LIN {X 0,Y 244.857,Z 831.109,A -85,B 0,C 180,E1 -23796.515,E2 -23796.515} C_VEL
LIN {X 0,Y 244.791,Z 831.344,A -85,B 0,C 180,E1 -23797.056,E2 -23797.056} C_VEL
LIN {X 0,Y 241.341,Z 845.058,A -85,B 0,C 180,E1 -23798.305,E2 -23798.305} C_VEL
LIN {X 0,Y 237.231,Z 858.218,A -85,B 0,C 180,E1 -23799.255,E2 -23799.255} C_VEL
LIN {X 0,Y 231.559,Z 871.694,A -85,B 0,C 180,E1 -23800.015,E2 -23800.015} C_VEL
LIN {X 0,Y 225.914,Z 882.984,A -85,B 0,C 180,E1 -23800.839,E2 -23800.839} C_VEL
LIN {X 0,Y 220.238,Z 892.764,A -85,B 0,C 180,E1 -23801.758,E2 -23801.758} C_VEL
LIN {X 0,Y 213.698,Z 902.652,A -85,B 0,C 180,E1 -23802.963,E2 -23802.963} C_VEL
LIN {X 0,Y 208.1,Z 910.323,A -85,B 0,C 180,E1 -23804.135,E2 -23804.135} C_VEL
LIN {X 0,Y 205.548,Z 913.56,A -85,B 0,C 180,E1 -23804.72,E2 -23804.72} C_VEL
LIN {X 0,Y 202.996,Z 916.447,A -85,B 0,C 180,E1 -23805.095,E2 -23805.095} C_VEL
LIN {X 0,Y 192.619,Z 924.938,A -85,B 0,C 180,E1 -23805.601,E2 -23805.601} C_VEL
LIN {X 0,Y 189.939,Z 927.241,A -85,B 0,C 180,E1 -23806.106,E2 -23806.106} C_VEL
LIN {X 0,Y 181.458,Z 935.069,A -85,B 0,C 180,E1 -23808.816,E2 -23808.816} C_VEL
LIN {X 0,Y 172.726,Z 942.329,A -85,B 0,C 180,E1 -23812.383,E2 -23812.383} C_VEL
LIN {X 0,Y 165.24,Z 947.878,A -85,B 0,C 180,E1 -23816.429,E2 -23816.429} C_VEL
LIN {X 0,Y 159.035,Z 952.034,A -85,B 0,C 180,E1 -23820.911,E2 -23820.911} C_VEL
LIN {X 0,Y 154.257,Z 954.977,A -85,B 0,C 180,E1 -23825.788,E2 -23825.788} C_VEL
LIN {X 0,Y 151.249,Z 956.558,A -85,B 0,C 180,E1 -23831.014,E2 -23831.014} C_VEL
LIN {X 0,Y 149.827,Z 956.906,A -85,B 0,C 180,E1 -23837.294,E2 -23837.294} C_VEL
LIN {X 0,Y 149.411,Z 960.982,A -85,B 0,C 180,E1 -23841.884,E2 -23841.884} C_VEL
LIN {X 0,Y 149.623,Z 962.776,A -85,B 0,C 180,E1 -23844.606,E2 -23844.606} C_VEL
LIN {X 0,Y 149.968,Z 964.104,A -85,B 0,C 180,E1 -23847.31,E2 -23847.31} C_VEL
LIN {X 0,Y 150.384,Z 964.99,A -85,B 0,C 180,E1 -23849.996,E2 -23849.996} C_VEL
LIN {X 0,Y 149.87,Z 965.286,A -85,B 0,C 180,E1 -23852.684,E2 -23852.684} C_VEL
LIN {X 0,Y 149.422,Z 965.12,A -85,B 0,C 180,E1 -23855.394,E2 -23855.394} C_VEL
LIN {X 0,Y 149.11,Z 964.525,A -85,B 0,C 180,E1 -23858.194,E2 -23858.194} C_VEL
LIN {X 0,Y 149.309,Z 962.242,A -85,B 0,C 180,E1 -23863.608,E2 -23863.608} C_VEL
LIN {X 0,Y 150.4,Z 959.454,A -85,B 0,C 180,E1 -23867.678,E2 -23867.678} C_VEL
LIN {X 0,Y 152.856,Z 954.714,A -85,B 0,C 180,E1 -23872.581,E2 -23872.581} C_VEL
LIN {X 0,Y 156.344,Z 949.182,A -85,B 0,C 180,E1 -23876.709,E2 -23876.709} C_VEL
LIN {X 0,Y 160.078,Z 942.88,A -85,B 0,C 180,E1 -23880.32,E2 -23880.32} C_VEL
LIN {X 0,Y 164.723,Z 935.183,A -85,B 0,C 180,E1 -23883.682,E2 -23883.682} C_VEL
LIN {X 0,Y 169.08,Z 927.436,A -85,B 0,C 180,E1 -23886.317,E2 -23886.317} C_VEL
LIN {X 0,Y 173.945,Z 918.156,A -85,B 0,C 180,E1 -23888.769,E2 -23888.769} C_VEL
LIN {X 0,Y 178.68,Z 907.985,A -85,B 0,C 180,E1 -23890.832,E2 -23890.832} C_VEL
LIN {X 0,Y 182.982,Z 896.807,A -85,B 0,C 180,E1 -23892.6,E2 -23892.6} C_VEL
LIN {X 0,Y 186.389,Z 886.413,A -85,B 0,C 180,E1 -23893.851,E2 -23893.851} C_VEL
LIN {X 0,Y 189.626,Z 874.101,A -85,B 0,C 180,E1 -23894.949,E2 -23894.949} C_VEL
LIN {X 0,Y 191.998,Z 861.503,A -85,B 0,C 180,E1 -23895.752,E2 -23895.752} C_VEL
LIN {X 0,Y 193.51,Z 846.926,A -85,B 0,C 180,E1 -23896.366,E2 -23896.366} C_VEL
LIN {X 0,Y 193.334,Z 821.886,A -85,B 0,C 180,E1 -23898.09,E2 -23898.09} C_VEL
LIN {X 0,Y 192.785,Z 805.817,A -85,B 0,C 180,E1 -23899.433,E2 -23899.433} C_VEL
LIN {X 0,Y 190.099,Z 798.147,A -85,B 0,C 180,E1 -23901.251,E2 -23901.251} C_VEL
LIN {X 0,Y 186.949,Z 790.152,A -85,B 0,C 180,E1 -23903.519,E2 -23903.519} C_VEL
LIN {X 0,Y 184.296,Z 784.188,A -85,B 0,C 180,E1 -23905.597,E2 -23905.597} C_VEL
LIN {X 0,Y 181.829,Z 778.84,A -85,B 0,C 180,E1 -23907.744,E2 -23907.744} C_VEL
LIN {X 0,Y 178.972,Z 772.86,A -85,B 0,C 180,E1 -23910.603,E2 -23910.603} C_VEL
LIN {X 0,Y 175.032,Z 765.017,A -85,B 0,C 180,E1 -23915.66,E2 -23915.66} C_VEL
LIN {X 0,Y 172.015,Z 759.221,A -85,B 0,C 180,E1 -23921.926,E2 -23921.926} C_VEL
LIN {X 0,Y 171.237,Z 756.818,A -85,B 0,C 180,E1 -23925.744,E2 -23925.744} C_VEL
LIN {X 0,Y 171.154,Z 756.438,A -85,B 0,C 180,E1 -23930.547,E2 -23930.547} C_VEL
LIN {X 0,Y 173.798,Z 758.074,A -85,B 0,C 180,E1 -23938.487,E2 -23938.487} C_VEL
LIN {X 0,Y 175.332,Z 761.318,A -85,B 0,C 180,E1 -23941.273,E2 -23941.273} C_VEL
LIN {X 0,Y 177.527,Z 763.638,A -85,B 0,C 180,E1 -23944.097,E2 -23944.097} C_VEL
LIN {X 0,Y 179.95,Z 767.21,A -85,B 0,C 180,E1 -23946.729,E2 -23946.729} C_VEL
LIN {X 0,Y 183.962,Z 773.224,A -85,B 0,C 180,E1 -23950.335,E2 -23950.335} C_VEL
LIN {X 0,Y 186.785,Z 777.685,A -85,B 0,C 180,E1 -23952.504,E2 -23952.504} C_VEL
LIN {X 0,Y 190.835,Z 784.368,A -85,B 0,C 180,E1 -23955.234,E2 -23955.234} C_VEL
LIN {X 0,Y 195.08,Z 792.248,A -85,B 0,C 180,E1 -23957.807,E2 -23957.807} C_VEL
LIN {X 0,Y 197.268,Z 796.713,A -85,B 0,C 180,E1 -23959.024,E2 -23959.024} C_VEL
LIN {X 0,Y 195.596,Z 824.391,A -85,B 0,C 180,E1 -23960.277,E2 -23960.277} C_VEL
LIN {X 0,Y 194.043,Z 837.391,A -85,B 0,C 180,E1 -23961.235,E2 -23961.235} C_VEL
LIN {X 0,Y 191.694,Z 849.84,A -85,B 0,C 180,E1 -23962.515,E2 -23962.515} C_VEL
LIN {X 0,Y 188.741,Z 860.968,A -85,B 0,C 180,E1 -23964.019,E2 -23964.019} C_VEL
LIN {X 0,Y 184.831,Z 872.603,A -85,B 0,C 180,E1 -23966.071,E2 -23966.071} C_VEL
LIN {X 0,Y 180.804,Z 882.425,A -85,B 0,C 180,E1 -23968.287,E2 -23968.287} C_VEL
LIN {X 0,Y 176.714,Z 890.906,A -85,B 0,C 180,E1 -23970.72,E2 -23970.72} C_VEL
LIN {X 0,Y 172.62,Z 898.364,A -85,B 0,C 180,E1 -23973.43,E2 -23973.43} C_VEL
LIN {X 0,Y 168.723,Z 904.617,A -85,B 0,C 180,E1 -23976.28,E2 -23976.28} C_VEL
LIN {X 0,Y 164.664,Z 910.533,A -85,B 0,C 180,E1 -23979.809,E2 -23979.809} C_VEL
LIN {X 0,Y 160.835,Z 915.42,A -85,B 0,C 180,E1 -23983.712,E2 -23983.712} C_VEL
LIN {X 0,Y 157.431,Z 919.174,A -85,B 0,C 180,E1 -23987.967,E2 -23987.967} C_VEL
LIN {X 0,Y 155.666,Z 920.852,A -85,B 0,C 180,E1 -23990.802,E2 -23990.802} C_VEL
LIN {X 0,Y 153.445,Z 922.533,A -85,B 0,C 180,E1 -23995.532,E2 -23995.532} C_VEL
LIN {X 0,Y 152.21,Z 922.921,A -85,B 0,C 180,E1 -23999.481,E2 -23999.481} C_VEL
LIN {X 0,Y 151.648,Z 922.674,A -85,B 0,C 180,E1 -24002.395,E2 -24002.395} C_VEL
LIN {X 0,Y 151.373,Z 921.923,A -85,B 0,C 180,E1 -24005.305,E2 -24005.305} C_VEL
LIN {X 0,Y 151.422,Z 920.718,A -85,B 0,C 180,E1 -24008.208,E2 -24008.208} C_VEL
LIN {X 0,Y 152.006,Z 918.04,A -85,B 0,C 180,E1 -24012.515,E2 -24012.515} C_VEL
LIN {X 0,Y 153.266,Z 914.247,A -85,B 0,C 180,E1 -24016.75,E2 -24016.75} C_VEL
LIN {X 0,Y 155.055,Z 909.269,A -85,B 0,C 180,E1 -24020.876,E2 -24020.876} C_VEL
LIN {X 0,Y 157.321,Z 902.95,A -85,B 0,C 180,E1 -24024.878,E2 -24024.878} C_VEL
LIN {X 0,Y 160.173,Z 895.068,A -85,B 0,C 180,E1 -24028.747,E2 -24028.747} C_VEL
LIN {X 0,Y 163.015,Z 886.699,A -85,B 0,C 180,E1 -24031.983,E2 -24031.983} C_VEL
LIN {X 0,Y 166.212,Z 876.183,A -85,B 0,C 180,E1 -24035.159,E2 -24035.159} C_VEL
LIN {X 0,Y 169.239,Z 864.857,A -85,B 0,C 180,E1 -24037.82,E2 -24037.82} C_VEL
LIN {X 0,Y 171.631,Z 854.357,A -85,B 0,C 180,E1 -24039.728,E2 -24039.728} C_VEL
LIN {X 0,Y 173.863,Z 841.585,A -85,B 0,C 180,E1 -24041.516,E2 -24041.516} C_VEL
LIN {X 0,Y 175.492,Z 828.533,A -85,B 0,C 180,E1 -24042.846,E2 -24042.846} C_VEL
LIN {X 0,Y 176.383,Z 815.217,A -85,B 0,C 180,E1 -24043.746,E2 -24043.746} C_VEL
LIN {X 0,Y 177.602,Z 782.378,A -85,B 0,C 180,E1 -24045.194,E2 -24045.194} C_VEL
LIN {X 0,Y 172.041,Z 770.25,A -85,B 0,C 180,E1 -24047.17,E2 -24047.17} C_VEL
LIN {X 0,Y 163.489,Z 754.986,A -85,B 0,C 180,E1 -24050.347,E2 -24050.347} C_VEL
LIN {X 0,Y 157.596,Z 745.662,A -85,B 0,C 180,E1 -24052.739,E2 -24052.739} C_VEL
LIN {X 0,Y 155.084,Z 741.988,A -85,B 0,C 180,E1 -24053.801,E2 -24053.801} C_VEL
LIN {X 0,Y 152.506,Z 738.118,A -85,B 0,C 180,E1 -24054.953,E2 -24054.953} C_VEL
LIN {X 0,Y 150.687,Z 735.478,A -85,B 0,C 180,E1 -24055.813,E2 -24055.813} C_VEL
LIN {X 0,Y 150.305,Z 734.187,A -85,B 0,C 180,E1 -24056.285,E2 -24056.285} C_VEL
LIN {X 0,Y 150.188,Z 733.748,A -85,B 0,C 180,E1 -24057.238,E2 -24057.238} C_VEL
LIN {X 0,Y 150.208,Z 733.739,A -85,B 0,C 180,E1 -24062.627,E2 -24062.627} C_VEL
LIN {X 0,Y 150.176,Z 733.747,A -85,B 0,C 180,E1 -24067.477,E2 -24067.477} C_VEL
LIN {X 0,Y 150.21,Z 733.927,A -85,B 0,C 180,E1 -24072.797,E2 -24072.797} C_VEL
LIN {X 0,Y 150.427,Z 734.862,A -85,B 0,C 180,E1 -24073.238,E2 -24073.238} C_VEL
LIN {X 0,Y 161.112,Z 767.276,A -85,B 0,C 180,E1 -24076.72,E2 -24076.72} C_VEL
LIN {X 0,Y 158.692,Z 816.623,A -85,B 0,C 180,E1 -24080.253,E2 -24080.253} C_VEL
LIN {X 0,Y 157.835,Z 828.145,A -85,B 0,C 180,E1 -24081.435,E2 -24081.435} C_VEL
LIN {X 0,Y 156.889,Z 838.329,A -85,B 0,C 180,E1 -24082.789,E2 -24082.789} C_VEL
LIN {X 0,Y 155.794,Z 848.57,A -85,B 0,C 180,E1 -24084.477,E2 -24084.477} C_VEL
LIN {X 0,Y 154.801,Z 857.302,A -85,B 0,C 180,E1 -24086.209,E2 -24086.209} C_VEL
LIN {X 0,Y 153.773,Z 866.172,A -85,B 0,C 180,E1 -24088.291,E2 -24088.291} C_VEL
LIN {X 0,Y 152.724,Z 874.335,A -85,B 0,C 180,E1 -24090.545,E2 -24090.545} C_VEL
LIN {X 0,Y 151.782,Z 882.385,A -85,B 0,C 180,E1 -24093.162,E2 -24093.162} C_VEL
LIN {X 0,Y 150.909,Z 891.404,A -85,B 0,C 180,E1 -24096.68,E2 -24096.68} C_VEL
LIN {X 0,Y 150.428,Z 898.5,A -85,B 0,C 180,E1 -24099.969,E2 -24099.969} C_VEL
LIN {X 0,Y 150.233,Z 904.129,A -85,B 0,C 180,E1 -24102.999,E2 -24102.999} C_VEL
LIN {X 0,Y 150.402,Z 909.603,A -85,B 0,C 180,E1 -24106.488,E2 -24106.488} C_VEL
LIN {X 0,Y 151.263,Z 914.934,A -85,B 0,C 180,E1 -24110.641,E2 -24110.641} C_VEL
LIN {X 0,Y 152.752,Z 919.142,A -85,B 0,C 180,E1 -24114.72,E2 -24114.72} C_VEL
LIN {X 0,Y 154.695,Z 922.06,A -85,B 0,C 180,E1 -24118.284,E2 -24118.284} C_VEL
LIN {X 0,Y 157.752,Z 924.553,A -85,B 0,C 180,E1 -24122.553,E2 -24122.553} C_VEL
LIN {X 0,Y 162.55,Z 926.08,A -85,B 0,C 180,E1 -24127.452,E2 -24127.452} C_VEL
LIN {X 0,Y 165.353,Z 926.213,A -85,B 0,C 180,E1 -24129.788,E2 -24129.788} C_VEL
LIN {X 0,Y 171.747,Z 925.212,A -85,B 0,C 180,E1 -24134.213,E2 -24134.213} C_VEL
LIN {X 0,Y 176.15,Z 923.903,A -85,B 0,C 180,E1 -24136.745,E2 -24136.745} C_VEL
LIN {X 0,Y 183.164,Z 920.704,A -85,B 0,C 180,E1 -24140.202,E2 -24140.202} C_VEL
LIN {X 0,Y 189.495,Z 916.99,A -85,B 0,C 180,E1 -24142.919,E2 -24142.919} C_VEL
LIN {X 0,Y 196.24,Z 912.131,A -85,B 0,C 180,E1 -24145.452,E2 -24145.452} C_VEL
LIN {X 0,Y 202.2,Z 907.143,A -85,B 0,C 180,E1 -24147.422,E2 -24147.422} C_VEL
LIN {X 0,Y 208.317,Z 901.17,A -85,B 0,C 180,E1 -24149.287,E2 -24149.287} C_VEL
LIN {X 0,Y 214.931,Z 893.757,A -85,B 0,C 180,E1 -24151.12,E2 -24151.12} C_VEL
LIN {X 0,Y 220.31,Z 886.741,A -85,B 0,C 180,E1 -24152.506,E2 -24152.506} C_VEL
LIN {X 0,Y 225.718,Z 878.716,A -85,B 0,C 180,E1 -24153.818,E2 -24153.818} C_VEL
LIN {X 0,Y 231.039,Z 869.384,A -85,B 0,C 180,E1 -24155.041,E2 -24155.041} C_VEL
LIN {X 0,Y 236.282,Z 858.337,A -85,B 0,C 180,E1 -24156.239,E2 -24156.239} C_VEL
LIN {X 0,Y 238.914,Z 851.646,A -85,B 0,C 180,E1 -24156.816,E2 -24156.816} C_VEL
LIN {X 0,Y 238.877,Z 851.821,A -85,B 0,C 180,E1 -24157.057,E2 -24157.057} C_VEL
LIN {X 0,Y 236.308,Z 858.808,A -85,B 0,C 180,E1 -24157.555,E2 -24157.555} C_VEL
LIN {X 0,Y 230.506,Z 871.836,A -85,B 0,C 180,E1 -24158.266,E2 -24158.266} C_VEL
LIN {X 0,Y 224.981,Z 882.268,A -85,B 0,C 180,E1 -24158.984,E2 -24158.984} C_VEL
LIN {X 0,Y 218.731,Z 892.42,A -85,B 0,C 180,E1 -24159.9,E2 -24159.9} C_VEL
LIN {X 0,Y 212.695,Z 901.133,A -85,B 0,C 180,E1 -24160.896,E2 -24160.896} C_VEL
LIN {X 0,Y 206.139,Z 909.58,A -85,B 0,C 180,E1 -24162.134,E2 -24162.134} C_VEL
LIN {X 0,Y 199.226,Z 917.636,A -85,B 0,C 180,E1 -24163.679,E2 -24163.679} C_VEL
LIN {X 0,Y 192.57,Z 924.669,A -85,B 0,C 180,E1 -24165.364,E2 -24165.364} C_VEL
LIN {X 0,Y 189.939,Z 927.241,A -85,B 0,C 180,E1 -24166.106,E2 -24166.106} C_VEL
LIN {X 0,Y 186.072,Z 930.673,A -85,B 0,C 180,E1 -24167.018,E2 -24167.018} C_VEL
LIN {X 0,Y 178.445,Z 935.858,A -85,B 0,C 180,E1 -24168.222,E2 -24168.222} C_VEL
LIN {X 0,Y 170.825,Z 940.29,A -85,B 0,C 180,E1 -24169.663,E2 -24169.663} C_VEL
LIN {X 0,Y 167.047,Z 942.549,A -85,B 0,C 180,E1 -24170.951,E2 -24170.951} C_VEL
LIN {X 0,Y 161.211,Z 946.474,A -85,B 0,C 180,E1 -24173.943,E2 -24173.943} C_VEL
LIN {X 0,Y 155.936,Z 949.734,A -85,B 0,C 180,E1 -24177.255,E2 -24177.255} C_VEL
LIN {X 0,Y 150.174,Z 952.868,A -85,B 0,C 180,E1 -24182.092,E2 -24182.092} C_VEL
LIN {X 0,Y 147.802,Z 953.95,A -85,B 0,C 180,E1 -24184.658,E2 -24184.658} C_VEL
LIN {X 0,Y 144.57,Z 955.216,A -85,B 0,C 180,E1 -24190.101,E2 -24190.101} C_VEL
LIN {X 0,Y 142.969,Z 955.384,A -85,B 0,C 180,E1 -24196.493,E2 -24196.493} C_VEL
LIN {X 0,Y 142.387,Z 959.731,A -85,B 0,C 180,E1 -24201.48,E2 -24201.48} C_VEL
LIN {X 0,Y 142.55,Z 961.596,A -85,B 0,C 180,E1 -24204.337,E2 -24204.337} C_VEL
LIN {X 0,Y 142.893,Z 962.963,A -85,B 0,C 180,E1 -24207.177,E2 -24207.177} C_VEL
LIN {X 0,Y 143.334,Z 963.887,A -85,B 0,C 180,E1 -24209.996,E2 -24209.996} C_VEL
LIN {X 0,Y 142.793,Z 964.216,A -85,B 0,C 180,E1 -24212.817,E2 -24212.817} C_VEL
LIN {X 0,Y 142.343,Z 964.109,A -85,B 0,C 180,E1 -24215.663,E2 -24215.663} C_VEL
LIN {X 0,Y 142.035,Z 963.562,A -85,B 0,C 180,E1 -24218.532,E2 -24218.532} C_VEL
LIN {X 0,Y 142.361,Z 961.325,A -85,B 0,C 180,E1 -24224.286,E2 -24224.286} C_VEL
LIN {X 0,Y 143.585,Z 958.615,A -85,B 0,C 180,E1 -24228.547,E2 -24228.547} C_VEL
LIN {X 0,Y 145.66,Z 954.974,A -85,B 0,C 180,E1 -24232.701,E2 -24232.701} C_VEL
LIN {X 0,Y 148.805,Z 950.346,A -85,B 0,C 180,E1 -24236.654,E2 -24236.654} C_VEL
LIN {X 0,Y 153.212,Z 943.497,A -85,B 0,C 180,E1 -24241.063,E2 -24241.063} C_VEL
LIN {X 0,Y 158.008,Z 936.183,A -85,B 0,C 180,E1 -24244.544,E2 -24244.544} C_VEL
LIN {X 0,Y 163.423,Z 927.179,A -85,B 0,C 180,E1 -24247.789,E2 -24247.789} C_VEL
LIN {X 0,Y 169.016,Z 917.092,A -85,B 0,C 180,E1 -24250.515,E2 -24250.515} C_VEL
LIN {X 0,Y 173.916,Z 906.962,A -85,B 0,C 180,E1 -24252.595,E2 -24252.595} C_VEL
LIN {X 0,Y 178.438,Z 895.826,A -85,B 0,C 180,E1 -24254.35,E2 -24254.35} C_VEL
LIN {X 0,Y 181.987,Z 885.454,A -85,B 0,C 180,E1 -24255.592,E2 -24255.592} C_VEL
LIN {X 0,Y 185.228,Z 873.548,A -85,B 0,C 180,E1 -24256.663,E2 -24256.663} C_VEL
LIN {X 0,Y 187.809,Z 860.468,A -85,B 0,C 180,E1 -24257.497,E2 -24257.497} C_VEL
LIN {X 0,Y 189.23,Z 847.787,A -85,B 0,C 180,E1 -24258.047,E2 -24258.047} C_VEL
LIN {X 0,Y 189.256,Z 823.547,A -85,B 0,C 180,E1 -24259.752,E2 -24259.752} C_VEL
LIN {X 0,Y 188.922,Z 808.906,A -85,B 0,C 180,E1 -24261.006,E2 -24261.006} C_VEL
LIN {X 0,Y 185.667,Z 799.516,A -85,B 0,C 180,E1 -24263.439,E2 -24263.439} C_VEL
LIN {X 0,Y 182.075,Z 790.42,A -85,B 0,C 180,E1 -24266.427,E2 -24266.427} C_VEL
LIN {X 0,Y 179.383,Z 784.402,A -85,B 0,C 180,E1 -24268.929,E2 -24268.929} C_VEL
LIN {X 0,Y 176.895,Z 778.825,A -85,B 0,C 180,E1 -24271.681,E2 -24271.681} C_VEL
LIN {X 0,Y 173.526,Z 771.565,A -85,B 0,C 180,E1 -24276.427,E2 -24276.427} C_VEL
LIN {X 0,Y 170.856,Z 765.951,A -85,B 0,C 180,E1 -24282.572,E2 -24282.572} C_VEL
LIN {X 0,Y 170.254,Z 763.802,A -85,B 0,C 180,E1 -24286.045,E2 -24286.045} C_VEL
LIN {X 0,Y 170.397,Z 763.591,A -85,B 0,C 180,E1 -24291.813,E2 -24291.813} C_VEL
LIN {X 0,Y 172.553,Z 764.994,A -85,B 0,C 180,E1 -24297.97,E2 -24297.97} C_VEL
LIN {X 0,Y 174.128,Z 768.299,A -85,B 0,C 180,E1 -24300.973,E2 -24300.973} C_VEL
LIN {X 0,Y 175.954,Z 770.323,A -85,B 0,C 180,E1 -24303.432,E2 -24303.432} C_VEL
LIN {X 0,Y 178.897,Z 774.892,A -85,B 0,C 180,E1 -24306.769,E2 -24306.769} C_VEL
LIN {X 0,Y 181.863,Z 779.533,A -85,B 0,C 180,E1 -24309.55,E2 -24309.55} C_VEL
LIN {X 0,Y 185.516,Z 785.499,A -85,B 0,C 180,E1 -24312.449,E2 -24312.449} C_VEL
LIN {X 0,Y 190.41,Z 794.409,A -85,B 0,C 180,E1 -24315.798,E2 -24315.798} C_VEL
LIN {X 0,Y 193.002,Z 799.778,A -85,B 0,C 180,E1 -24317.418,E2 -24317.418} C_VEL
LIN {X 0,Y 191.339,Z 825.631,A -85,B 0,C 180,E1 -24318.63,E2 -24318.63} C_VEL
LIN {X 0,Y 189.639,Z 839.007,A -85,B 0,C 180,E1 -24319.64,E2 -24319.64} C_VEL
LIN {X 0,Y 187.173,Z 851.209,A -85,B 0,C 180,E1 -24320.914,E2 -24320.914} C_VEL
LIN {X 0,Y 183.996,Z 862.479,A -85,B 0,C 180,E1 -24322.456,E2 -24322.456} C_VEL
LIN {X 0,Y 180.29,Z 873.055,A -85,B 0,C 180,E1 -24324.338,E2 -24324.338} C_VEL
LIN {X 0,Y 176.046,Z 882.97,A -85,B 0,C 180,E1 -24326.568,E2 -24326.568} C_VEL
LIN {X 0,Y 171.264,Z 892.376,A -85,B 0,C 180,E1 -24329.309,E2 -24329.309} C_VEL
LIN {X 0,Y 166.475,Z 900.52,A -85,B 0,C 180,E1 -24332.407,E2 -24332.407} C_VEL
LIN {X 0,Y 162.055,Z 907.056,A -85,B 0,C 180,E1 -24335.602,E2 -24335.602} C_VEL
LIN {X 0,Y 157.839,Z 912.736,A -85,B 0,C 180,E1 -24339.291,E2 -24339.291} C_VEL
LIN {X 0,Y 153.986,Z 917.204,A -85,B 0,C 180,E1 -24343.206,E2 -24343.206} C_VEL
LIN {X 0,Y 151.683,Z 919.544,A -85,B 0,C 180,E1 -24345.979,E2 -24345.979} C_VEL
LIN {X 0,Y 149.656,Z 921.439,A -85,B 0,C 180,E1 -24348.9,E2 -24348.9} C_VEL
LIN {X 0,Y 147.959,Z 922.759,A -85,B 0,C 180,E1 -24351.872,E2 -24351.872} C_VEL
LIN {X 0,Y 146.615,Z 923.598,A -85,B 0,C 180,E1 -24354.89,E2 -24354.89} C_VEL
LIN {X 0,Y 145.575,Z 923.958,A -85,B 0,C 180,E1 -24357.929,E2 -24357.929} C_VEL
LIN {X 0,Y 144.831,Z 923.822,A -85,B 0,C 180,E1 -24360.976,E2 -24360.976} C_VEL
LIN {X 0,Y 144.416,Z 923.251,A -85,B 0,C 180,E1 -24364.029,E2 -24364.029} C_VEL
LIN {X 0,Y 144.361,Z 921.921,A -85,B 0,C 180,E1 -24367.668,E2 -24367.668} C_VEL
LIN {X 0,Y 145.083,Z 918.687,A -85,B 0,C 180,E1 -24373.108,E2 -24373.108} C_VEL
LIN {X 0,Y 146.441,Z 914.74,A -85,B 0,C 180,E1 -24377.532,E2 -24377.532} C_VEL
LIN {X 0,Y 148.376,Z 909.584,A -85,B 0,C 180,E1 -24381.835,E2 -24381.835} C_VEL
LIN {X 0,Y 150.838,Z 903.098,A -85,B 0,C 180,E1 -24385.996,E2 -24385.996} C_VEL
LIN {X 0,Y 153.888,Z 895.031,A -85,B 0,C 180,E1 -24390.004,E2 -24390.004} C_VEL
LIN {X 0,Y 156.754,Z 886.775,A -85,B 0,C 180,E1 -24393.217,E2 -24393.217} C_VEL
LIN {X 0,Y 159.938,Z 876.714,A -85,B 0,C 180,E1 -24396.311,E2 -24396.311} C_VEL
LIN {X 0,Y 162.815,Z 866.371,A -85,B 0,C 180,E1 -24398.818,E2 -24398.818} C_VEL
LIN {X 0,Y 165.688,Z 854.358,A -85,B 0,C 180,E1 -24401.047,E2 -24401.047} C_VEL
LIN {X 0,Y 167.901,Z 842.082,A -85,B 0,C 180,E1 -24402.79,E2 -24402.79} C_VEL
LIN {X 0,Y 169.575,Z 829.05,A -85,B 0,C 180,E1 -24404.134,E2 -24404.134} C_VEL
LIN {X 0,Y 170.521,Z 815.506,A -85,B 0,C 180,E1 -24405.055,E2 -24405.055} C_VEL
LIN {X 0,Y 171.772,Z 784.662,A -85,B 0,C 180,E1 -24406.448,E2 -24406.448} C_VEL
LIN {X 0,Y 166.895,Z 773.878,A -85,B 0,C 180,E1 -24408.295,E2 -24408.295} C_VEL
LIN {X 0,Y 158.208,Z 758.184,A -85,B 0,C 180,E1 -24411.745,E2 -24411.745} C_VEL
LIN {X 0,Y 151.544,Z 747.775,A -85,B 0,C 180,E1 -24414.639,E2 -24414.639} C_VEL
LIN {X 0,Y 148.161,Z 742.893,A -85,B 0,C 180,E1 -24416.227,E2 -24416.227} C_VEL
LIN {X 0,Y 145.883,Z 739.368,A -85,B 0,C 180,E1 -24417.383,E2 -24417.383} C_VEL
LIN {X 0,Y 143.969,Z 737.259,A -85,B 0,C 180,E1 -24418.336,E2 -24418.336} C_VEL
LIN {X 0,Y 143.173,Z 735.183,A -85,B 0,C 180,E1 -24419.065,E2 -24419.065} C_VEL
LIN {X 0,Y 143.096,Z 734.694,A -85,B 0,C 180,E1 -24419.825,E2 -24419.825} C_VEL
LIN {X 0,Y 143.14,Z 734.61,A -85,B 0,C 180,E1 -24423.416,E2 -24423.416} C_VEL
LIN {X 0,Y 143.065,Z 734.665,A -85,B 0,C 180,E1 -24429.694,E2 -24429.694} C_VEL
LIN {X 0,Y 143.169,Z 734.859,A -85,B 0,C 180,E1 -24432.164,E2 -24432.164} C_VEL
LIN {X 0,Y 143.327,Z 735.632,A -85,B 0,C 180,E1 -24432.545,E2 -24432.545} C_VEL
LIN {X 0,Y 154.136,Z 768.162,A -85,B 0,C 180,E1 -24436.231,E2 -24436.231} C_VEL
LIN {X 0,Y 151.652,Z 816.898,A -85,B 0,C 180,E1 -24439.874,E2 -24439.874} C_VEL
LIN {X 0,Y 150.738,Z 829.345,A -85,B 0,C 180,E1 -24441.206,E2 -24441.206} C_VEL
LIN {X 0,Y 149.781,Z 839.313,A -85,B 0,C 180,E1 -24442.598,E2 -24442.598} C_VEL
LIN {X 0,Y 148.649,Z 849.364,A -85,B 0,C 180,E1 -24444.341,E2 -24444.341} C_VEL
LIN {X 0,Y 147.539,Z 859.005,A -85,B 0,C 180,E1 -24446.374,E2 -24446.374} C_VEL
LIN {X 0,Y 146.39,Z 868.536,A -85,B 0,C 180,E1 -24448.788,E2 -24448.788} C_VEL
LIN {X 0,Y 145.249,Z 877.393,A -85,B 0,C 180,E1 -24451.457,E2 -24451.457} C_VEL
LIN {X 0,Y 144.441,Z 884.715,A -85,B 0,C 180,E1 -24454.029,E2 -24454.029} C_VEL
LIN {X 0,Y 143.651,Z 892.968,A -85,B 0,C 180,E1 -24457.44,E2 -24457.44} C_VEL
LIN {X 0,Y 143.273,Z 899.543,A -85,B 0,C 180,E1 -24460.663,E2 -24460.663} C_VEL
LIN {X 0,Y 143.14,Z 905.903,A -85,B 0,C 180,E1 -24464.333,E2 -24464.333} C_VEL
LIN {X 0,Y 143.575,Z 911.628,A -85,B 0,C 180,E1 -24468.256,E2 -24468.256} C_VEL
LIN {X 0,Y 144.411,Z 915.811,A -85,B 0,C 180,E1 -24471.604,E2 -24471.604} C_VEL
LIN {X 0,Y 146.117,Z 920.106,A -85,B 0,C 180,E1 -24475.862,E2 -24475.862} C_VEL
LIN {X 0,Y 148.485,Z 923.397,A -85,B 0,C 180,E1 -24480,E2 -24480} C_VEL
LIN {X 0,Y 152.814,Z 926.294,A -85,B 0,C 180,E1 -24485.277,E2 -24485.277} C_VEL
LIN {X 0,Y 156.431,Z 927.329,A -85,B 0,C 180,E1 -24488.714,E2 -24488.714} C_VEL
LIN {X 0,Y 161.463,Z 927.53,A -85,B 0,C 180,E1 -24492.57,E2 -24492.57} C_VEL
LIN {X 0,Y 164.908,Z 927.235,A -85,B 0,C 180,E1 -24494.815,E2 -24494.815} C_VEL
LIN {X 0,Y 172.527,Z 925.233,A -85,B 0,C 180,E1 -24499.019,E2 -24499.019} C_VEL
LIN {X 0,Y 178.85,Z 922.67,A -85,B 0,C 180,E1 -24501.919,E2 -24501.919} C_VEL
LIN {X 0,Y 185.553,Z 919.115,A -85,B 0,C 180,E1 -24504.622,E2 -24504.622} C_VEL
LIN {X 0,Y 192.667,Z 914.465,A -85,B 0,C 180,E1 -24507.127,E2 -24507.127} C_VEL
LIN {X 0,Y 200.161,Z 908.58,A -85,B 0,C 180,E1 -24509.443,E2 -24509.443} C_VEL
LIN {X 0,Y 205.326,Z 903.977,A -85,B 0,C 180,E1 -24510.892,E2 -24510.892} C_VEL
LIN {X 0,Y 211.943,Z 897.119,A -85,B 0,C 180,E1 -24512.605,E2 -24512.605} C_VEL
LIN {X 0,Y 218.691,Z 888.993,A -85,B 0,C 180,E1 -24514.221,E2 -24514.221} C_VEL
LIN {X 0,Y 224.581,Z 880.679,A -85,B 0,C 180,E1 -24515.543,E2 -24515.543} C_VEL
LIN {X 0,Y 228.365,Z 874.777,A -85,B 0,C 180,E1 -24516.316,E2 -24516.316} C_VEL
LIN {X 0,Y 227.941,Z 875.72,A -85,B 0,C 180,E1 -24516.709,E2 -24516.709} C_VEL
LIN {X 0,Y 220.701,Z 887.61,A -85,B 0,C 180,E1 -24517.59,E2 -24517.59} C_VEL
LIN {X 0,Y 213.56,Z 897.825,A -85,B 0,C 180,E1 -24518.59,E2 -24518.59} C_VEL
LIN {X 0,Y 205.949,Z 907.304,A -85,B 0,C 180,E1 -24519.838,E2 -24519.838} C_VEL
LIN {X 0,Y 198.644,Z 915.456,A -85,B 0,C 180,E1 -24521.247,E2 -24521.247} C_VEL
LIN {X 0,Y 190.336,Z 923.726,A -85,B 0,C 180,E1 -24523.172,E2 -24523.172} C_VEL
LIN {X 0,Y 182.45,Z 930.784,A -85,B 0,C 180,E1 -24525.328,E2 -24525.328} C_VEL
LIN {X 0,Y 176.206,Z 935.857,A -85,B 0,C 180,E1 -24527.304,E2 -24527.304} C_VEL
LIN {X 0,Y 169.372,Z 941.038,A -85,B 0,C 180,E1 -24529.968,E2 -24529.968} C_VEL
LIN {X 0,Y 167.047,Z 942.549,A -85,B 0,C 180,E1 -24530.951,E2 -24530.951} C_VEL
LIN {X 0,Y 163.342,Z 944.808,A -85,B 0,C 180,E1 -24532.373,E2 -24532.373} C_VEL
LIN {X 0,Y 156.022,Z 947.759,A -85,B 0,C 180,E1 -24534.534,E2 -24534.534} C_VEL
LIN {X 0,Y 149.043,Z 950.012,A -85,B 0,C 180,E1 -24537.006,E2 -24537.006} C_VEL
LIN {X 0,Y 145.961,Z 951.091,A -85,B 0,C 180,E1 -24538.897,E2 -24538.897} C_VEL
LIN {X 0,Y 141.458,Z 952.873,A -85,B 0,C 180,E1 -24543.435,E2 -24543.435} C_VEL
LIN {X 0,Y 137.959,Z 953.774,A -85,B 0,C 180,E1 -24549.104,E2 -24549.104} C_VEL
LIN {X 0,Y 136.212,Z 953.695,A -85,B 0,C 180,E1 -24555.427,E2 -24555.427} C_VEL
LIN {X 0,Y 135.363,Z 958.478,A -85,B 0,C 180,E1 -24561.035,E2 -24561.035} C_VEL
LIN {X 0,Y 135.486,Z 960.401,A -85,B 0,C 180,E1 -24564.041,E2 -24564.041} C_VEL
LIN {X 0,Y 135.815,Z 961.821,A -85,B 0,C 180,E1 -24567.029,E2 -24567.029} C_VEL
LIN {X 0,Y 136.281,Z 962.784,A -85,B 0,C 180,E1 -24569.996,E2 -24569.996} C_VEL
LIN {X 0,Y 135.716,Z 963.141,A -85,B 0,C 180,E1 -24572.964,E2 -24572.964} C_VEL
LIN {X 0,Y 135.269,Z 963.082,A -85,B 0,C 180,E1 -24575.96,E2 -24575.96} C_VEL
LIN {X 0,Y 134.959,Z 962.58,A -85,B 0,C 180,E1 -24578.983,E2 -24578.983} C_VEL
LIN {X 0,Y 135.426,Z 960.421,A -85,B 0,C 180,E1 -24585.034,E2 -24585.034} C_VEL
LIN {X 0,Y 137.451,Z 956.728,A -85,B 0,C 180,E1 -24590.967,E2 -24590.967} C_VEL
LIN {X 0,Y 140.637,Z 952.106,A -85,B 0,C 180,E1 -24595.907,E2 -24595.907} C_VEL
LIN {X 0,Y 145.011,Z 946.036,A -85,B 0,C 180,E1 -24600.585,E2 -24600.585} C_VEL
LIN {X 0,Y 149.608,Z 939.556,A -85,B 0,C 180,E1 -24604.308,E2 -24604.308} C_VEL
LIN {X 0,Y 154.922,Z 931.632,A -85,B 0,C 180,E1 -24607.76,E2 -24607.76} C_VEL
LIN {X 0,Y 160.973,Z 921.826,A -85,B 0,C 180,E1 -24610.906,E2 -24610.906} C_VEL
LIN {X 0,Y 166.428,Z 911.816,A -85,B 0,C 180,E1 -24613.326,E2 -24613.326} C_VEL
LIN {X 0,Y 171.712,Z 900.711,A -85,B 0,C 180,E1 -24615.322,E2 -24615.322} C_VEL
LIN {X 0,Y 176.473,Z 888.208,A -85,B 0,C 180,E1 -24617.03,E2 -24617.03} C_VEL
LIN {X 0,Y 180.445,Z 875.336,A -85,B 0,C 180,E1 -24618.273,E2 -24618.273} C_VEL
LIN {X 0,Y 183.303,Z 862.327,A -85,B 0,C 180,E1 -24619.166,E2 -24619.166} C_VEL
LIN {X 0,Y 185.162,Z 848.476,A -85,B 0,C 180,E1 -24619.816,E2 -24619.816} C_VEL
LIN {X 0,Y 185.39,Z 823.806,A -85,B 0,C 180,E1 -24621.611,E2 -24621.611} C_VEL
LIN {X 0,Y 185.162,Z 811.985,A -85,B 0,C 180,E1 -24622.68,E2 -24622.68} C_VEL
LIN {X 0,Y 182.198,Z 803.163,A -85,B 0,C 180,E1 -24625.144,E2 -24625.144} C_VEL
LIN {X 0,Y 179.277,Z 795.408,A -85,B 0,C 180,E1 -24627.836,E2 -24627.836} C_VEL
LIN {X 0,Y 177.126,Z 790.119,A -85,B 0,C 180,E1 -24630.081,E2 -24630.081} C_VEL
LIN {X 0,Y 174.907,Z 784.791,A -85,B 0,C 180,E1 -24632.76,E2 -24632.76} C_VEL
LIN {X 0,Y 172.06,Z 778.126,A -85,B 0,C 180,E1 -24637.191,E2 -24637.191} C_VEL
LIN {X 0,Y 169.734,Z 772.737,A -85,B 0,C 180,E1 -24643.152,E2 -24643.152} C_VEL
LIN {X 0,Y 169.267,Z 770.797,A -85,B 0,C 180,E1 -24646.395,E2 -24646.395} C_VEL
LIN {X 0,Y 169.435,Z 770.624,A -85,B 0,C 180,E1 -24651.721,E2 -24651.721} C_VEL
LIN {X 0,Y 171.347,Z 771.955,A -85,B 0,C 180,E1 -24657.503,E2 -24657.503} C_VEL
LIN {X 0,Y 172.777,Z 775.071,A -85,B 0,C 180,E1 -24660.429,E2 -24660.429} C_VEL
LIN {X 0,Y 174.41,Z 776.988,A -85,B 0,C 180,E1 -24662.758,E2 -24662.758} C_VEL
LIN {X 0,Y 176.992,Z 781.232,A -85,B 0,C 180,E1 -24665.912,E2 -24665.912} C_VEL
LIN {X 0,Y 180.068,Z 786.304,A -85,B 0,C 180,E1 -24668.982,E2 -24668.982} C_VEL
LIN {X 0,Y 183.743,Z 792.756,A -85,B 0,C 180,E1 -24672.037,E2 -24672.037} C_VEL
LIN {X 0,Y 187.494,Z 799.963,A -85,B 0,C 180,E1 -24674.766,E2 -24674.766} C_VEL
LIN {X 0,Y 188.959,Z 803.066,A -85,B 0,C 180,E1 -24675.751,E2 -24675.751} C_VEL
LIN {X 0,Y 187.321,Z 826.875,A -85,B 0,C 180,E1 -24676.902,E2 -24676.902} C_VEL
LIN {X 0,Y 185.498,Z 840.254,A -85,B 0,C 180,E1 -24677.929,E2 -24677.929} C_VEL
LIN {X 0,Y 182.822,Z 852.627,A -85,B 0,C 180,E1 -24679.237,E2 -24679.237} C_VEL
LIN {X 0,Y 179.593,Z 863.493,A -85,B 0,C 180,E1 -24680.738,E2 -24680.738} C_VEL
LIN {X 0,Y 175.341,Z 874.949,A -85,B 0,C 180,E1 -24682.807,E2 -24682.807} C_VEL
LIN {X 0,Y 170.774,Z 884.972,A -85,B 0,C 180,E1 -24685.134,E2 -24685.134} C_VEL
LIN {X 0,Y 165.464,Z 894.675,A -85,B 0,C 180,E1 -24688.083,E2 -24688.083} C_VEL
LIN {X 0,Y 160.635,Z 902.354,A -85,B 0,C 180,E1 -24691.144,E2 -24691.144} C_VEL
LIN {X 0,Y 155.787,Z 909.025,A -85,B 0,C 180,E1 -24694.59,E2 -24694.59} C_VEL
LIN {X 0,Y 151.723,Z 914.055,A -85,B 0,C 180,E1 -24698.058,E2 -24698.058} C_VEL
LIN {X 0,Y 148.046,Z 918.026,A -85,B 0,C 180,E1 -24701.653,E2 -24701.653} C_VEL
LIN {X 0,Y 144.933,Z 920.984,A -85,B 0,C 180,E1 -24705.328,E2 -24705.328} C_VEL
LIN {X 0,Y 141.888,Z 923.45,A -85,B 0,C 180,E1 -24709.921,E2 -24709.921} C_VEL
LIN {X 0,Y 140.184,Z 924.482,A -85,B 0,C 180,E1 -24713.337,E2 -24713.337} C_VEL
LIN {X 0,Y 139.031,Z 924.925,A -85,B 0,C 180,E1 -24716.222,E2 -24716.222} C_VEL
LIN {X 0,Y 138.018,Z 924.904,A -85,B 0,C 180,E1 -24719.959,E2 -24719.959} C_VEL
LIN {X 0,Y 137.314,Z 923.597,A -85,B 0,C 180,E1 -24725.834,E2 -24725.834} C_VEL
LIN {X 0,Y 137.389,Z 922.23,A -85,B 0,C 180,E1 -24729.023,E2 -24729.023} C_VEL
LIN {X 0,Y 138.429,Z 918.519,A -85,B 0,C 180,E1 -24734.717,E2 -24734.717} C_VEL
LIN {X 0,Y 140.272,Z 913.573,A -85,B 0,C 180,E1 -24739.905,E2 -24739.905} C_VEL
LIN {X 0,Y 142.532,Z 907.832,A -85,B 0,C 180,E1 -24744.345,E2 -24744.345} C_VEL
LIN {X 0,Y 145.43,Z 900.643,A -85,B 0,C 180,E1 -24748.62,E2 -24748.62} C_VEL
LIN {X 0,Y 148.419,Z 892.912,A -85,B 0,C 180,E1 -24752.221,E2 -24752.221} C_VEL
LIN {X 0,Y 151.7,Z 883.558,A -85,B 0,C 180,E1 -24755.654,E2 -24755.654} C_VEL
LIN {X 0,Y 155.214,Z 872.472,A -85,B 0,C 180,E1 -24758.794,E2 -24758.794} C_VEL
LIN {X 0,Y 157.793,Z 862.94,A -85,B 0,C 180,E1 -24760.921,E2 -24760.921} C_VEL
LIN {X 0,Y 160.501,Z 851.147,A -85,B 0,C 180,E1 -24762.972,E2 -24762.972} C_VEL
LIN {X 0,Y 162.576,Z 839.066,A -85,B 0,C 180,E1 -24764.556,E2 -24764.556} C_VEL
LIN {X 0,Y 164.092,Z 825.529,A -85,B 0,C 180,E1 -24765.847,E2 -24765.847} C_VEL
LIN {X 0,Y 164.888,Z 810.544,A -85,B 0,C 180,E1 -24766.727,E2 -24766.727} C_VEL
LIN {X 0,Y 165.913,Z 786.671,A -85,B 0,C 180,E1 -24767.822,E2 -24767.822} C_VEL
LIN {X 0,Y 161.561,Z 777.052,A -85,B 0,C 180,E1 -24769.573,E2 -24769.573} C_VEL
LIN {X 0,Y 153.77,Z 762.826,A -85,B 0,C 180,E1 -24772.874,E2 -24772.874} C_VEL
LIN {X 0,Y 147.701,Z 753.099,A -85,B 0,C 180,E1 -24775.675,E2 -24775.675} C_VEL
LIN {X 0,Y 142.161,Z 744.883,A -85,B 0,C 180,E1 -24778.525,E2 -24778.525} C_VEL
LIN {X 0,Y 139.798,Z 741.665,A -85,B 0,C 180,E1 -24779.826,E2 -24779.826} C_VEL
LIN {X 0,Y 138.996,Z 740.432,A -85,B 0,C 180,E1 -24780.291,E2 -24780.291} C_VEL
LIN {X 0,Y 136.946,Z 738.037,A -85,B 0,C 180,E1 -24781.443,E2 -24781.443} C_VEL
LIN {X 0,Y 136.236,Z 736.135,A -85,B 0,C 180,E1 -24782.16,E2 -24782.16} C_VEL
LIN {X 0,Y 136.129,Z 735.51,A -85,B 0,C 180,E1 -24783.182,E2 -24783.182} C_VEL
LIN {X 0,Y 136.092,Z 735.539,A -85,B 0,C 180,E1 -24790.814,E2 -24790.814} C_VEL
LIN {X 0,Y 136.171,Z 735.909,A -85,B 0,C 180,E1 -24791.576,E2 -24791.576} C_VEL
LIN {X 0,Y 136.585,Z 737.479,A -85,B 0,C 180,E1 -24791.989,E2 -24791.989} C_VEL
LIN {X 0,Y 147.136,Z 769.241,A -85,B 0,C 180,E1 -24795.716,E2 -24795.716} C_VEL
LIN {X 0,Y 144.558,Z 818.678,A -85,B 0,C 180,E1 -24799.667,E2 -24799.667} C_VEL
LIN {X 0,Y 143.554,Z 830.387,A -85,B 0,C 180,E1 -24801,E2 -24801} C_VEL
LIN {X 0,Y 142.574,Z 840.809,A -85,B 0,C 180,E1 -24802.546,E2 -24802.546} C_VEL
LIN {X 0,Y 141.472,Z 850.35,A -85,B 0,C 180,E1 -24804.287,E2 -24804.287} C_VEL
LIN {X 0,Y 140.272,Z 860.558,A -85,B 0,C 180,E1 -24806.555,E2 -24806.555} C_VEL
LIN {X 0,Y 139.138,Z 869.649,A -85,B 0,C 180,E1 -24808.979,E2 -24808.979} C_VEL
LIN {X 0,Y 138.097,Z 877.67,A -85,B 0,C 180,E1 -24811.502,E2 -24811.502} C_VEL
LIN {X 0,Y 137.312,Z 885.07,A -85,B 0,C 180,E1 -24814.211,E2 -24814.211} C_VEL
LIN {X 0,Y 136.527,Z 893.619,A -85,B 0,C 180,E1 -24817.919,E2 -24817.919} C_VEL
LIN {X 0,Y 136.153,Z 900.059,A -85,B 0,C 180,E1 -24821.178,E2 -24821.178} C_VEL
LIN {X 0,Y 136.095,Z 906.551,A -85,B 0,C 180,E1 -24825.036,E2 -24825.036} C_VEL
LIN {X 0,Y 136.763,Z 912.956,A -85,B 0,C 180,E1 -24829.663,E2 -24829.663} C_VEL
LIN {X 0,Y 138.142,Z 918.092,A -85,B 0,C 180,E1 -24834.16,E2 -24834.16} C_VEL
LIN {X 0,Y 139.537,Z 921.032,A -85,B 0,C 180,E1 -24837.113,E2 -24837.113} C_VEL
LIN {X 0,Y 143.184,Z 925.256,A -85,B 0,C 180,E1 -24842.813,E2 -24842.813} C_VEL
LIN {X 0,Y 145.579,Z 926.872,A -85,B 0,C 180,E1 -24845.54,E2 -24845.54} C_VEL
LIN {X 0,Y 151.195,Z 928.701,A -85,B 0,C 180,E1 -24850.715,E2 -24850.715} C_VEL
LIN {X 0,Y 154.488,Z 929.031,A -85,B 0,C 180,E1 -24853.147,E2 -24853.147} C_VEL
LIN {X 0,Y 162.786,Z 928.279,A -85,B 0,C 180,E1 -24858.219,E2 -24858.219} C_VEL
LIN {X 0,Y 170.204,Z 926.267,A -85,B 0,C 180,E1 -24861.816,E2 -24861.816} C_VEL
LIN {X 0,Y 174.717,Z 924.672,A -85,B 0,C 180,E1 -24863.719,E2 -24863.719} C_VEL
LIN {X 0,Y 180.811,Z 921.824,A -85,B 0,C 180,E1 -24866.043,E2 -24866.043} C_VEL
LIN {X 0,Y 189.277,Z 916.88,A -85,B 0,C 180,E1 -24868.862,E2 -24868.862} C_VEL
LIN {X 0,Y 198.308,Z 910.213,A -85,B 0,C 180,E1 -24871.455,E2 -24871.455} C_VEL
LIN {X 0,Y 205.239,Z 904.244,A -85,B 0,C 180,E1 -24873.222,E2 -24873.222} C_VEL
LIN {X 0,Y 210.813,Z 898.734,A -85,B 0,C 180,E1 -24874.523,E2 -24874.523} C_VEL
LIN {X 0,Y 216.638,Z 892.244,A -85,B 0,C 180,E1 -24875.799,E2 -24875.799} C_VEL
LIN {X 0,Y 217.315,Z 891.423,A -85,B 0,C 180,E1 -24876.046,E2 -24876.046} C_VEL
LIN {X 0,Y 208.044,Z 903.165,A -85,B 0,C 180,E1 -24877.289,E2 -24877.289} C_VEL
LIN {X 0,Y 200.055,Z 911.949,A -85,B 0,C 180,E1 -24878.584,E2 -24878.584} C_VEL
LIN {X 0,Y 191.266,Z 920.433,A -85,B 0,C 180,E1 -24880.315,E2 -24880.315} C_VEL
LIN {X 0,Y 182.852,Z 927.716,A -85,B 0,C 180,E1 -24882.274,E2 -24882.274} C_VEL
LIN {X 0,Y 173.606,Z 934.749,A -85,B 0,C 180,E1 -24884.887,E2 -24884.887} C_VEL
LIN {X 0,Y 166.274,Z 939.796,A -85,B 0,C 180,E1 -24887.442,E2 -24887.442} C_VEL
LIN {X 0,Y 159.593,Z 944.002,A -85,B 0,C 180,E1 -24890.313,E2 -24890.313} C_VEL
LIN {X 0,Y 153.608,Z 947.376,A -85,B 0,C 180,E1 -24893.498,E2 -24893.498} C_VEL
LIN {X 0,Y 145.961,Z 951.091,A -85,B 0,C 180,E1 -24898.897,E2 -24898.897} C_VEL
LIN {X 0,Y 143.11,Z 951.994,A -85,B 0,C 180,E1 -24900.924,E2 -24900.924} C_VEL
LIN {X 0,Y 137.327,Z 952.628,A -85,B 0,C 180,E1 -24904.207,E2 -24904.207} C_VEL
LIN {X 0,Y 132.218,Z 952.361,A -85,B 0,C 180,E1 -24907.805,E2 -24907.805} C_VEL
LIN {X 0,Y 130.503,Z 952.16,A -85,B 0,C 180,E1 -24910.262,E2 -24910.262} C_VEL
LIN {X 0,Y 129.483,Z 951.942,A -85,B 0,C 180,E1 -24914.248,E2 -24914.248} C_VEL
LIN {X 0,Y 128.442,Z 956.076,A -85,B 0,C 180,E1 -24918.956,E2 -24918.956} C_VEL
LIN {X 0,Y 128.429,Z 959.177,A -85,B 0,C 180,E1 -24923.712,E2 -24923.712} C_VEL
LIN {X 0,Y 128.739,Z 960.672,A -85,B 0,C 180,E1 -24926.866,E2 -24926.866} C_VEL
LIN {X 0,Y 129.224,Z 961.675,A -85,B 0,C 180,E1 -24929.995,E2 -24929.995} C_VEL
LIN {X 0,Y 128.638,Z 962.062,A -85,B 0,C 180,E1 -24933.127,E2 -24933.127} C_VEL
LIN {X 0,Y 127.946,Z 961.736,A -85,B 0,C 180,E1 -24938.612,E2 -24938.612} C_VEL
LIN {X 0,Y 127.999,Z 960.745,A -85,B 0,C 180,E1 -24942.682,E2 -24942.682} C_VEL
LIN {X 0,Y 129.418,Z 957.906,A -85,B 0,C 180,E1 -24949.011,E2 -24949.011} C_VEL
LIN {X 0,Y 131.6,Z 954.743,A -85,B 0,C 180,E1 -24953.606,E2 -24953.606} C_VEL
LIN {X 0,Y 134.898,Z 950.644,A -85,B 0,C 180,E1 -24957.957,E2 -24957.957} C_VEL
LIN {X 0,Y 138.907,Z 945.47,A -85,B 0,C 180,E1 -24962.084,E2 -24962.084} C_VEL
LIN {X 0,Y 143.79,Z 939.1,A -85,B 0,C 180,E1 -24965.905,E2 -24965.905} C_VEL
LIN {X 0,Y 149.356,Z 931.309,A -85,B 0,C 180,E1 -24969.433,E2 -24969.433} C_VEL
LIN {X 0,Y 154.571,Z 923.466,A -85,B 0,C 180,E1 -24972.111,E2 -24972.111} C_VEL
LIN {X 0,Y 160.787,Z 913.002,A -85,B 0,C 180,E1 -24974.81,E2 -24974.81} C_VEL
LIN {X 0,Y 166.188,Z 902.449,A -85,B 0,C 180,E1 -24976.838,E2 -24976.838} C_VEL
LIN {X 0,Y 171.084,Z 890.846,A -85,B 0,C 180,E1 -24978.558,E2 -24978.558} C_VEL
LIN {X 0,Y 175.358,Z 878.607,A -85,B 0,C 180,E1 -24979.825,E2 -24979.825} C_VEL
LIN {X 0,Y 178.68,Z 865.731,A -85,B 0,C 180,E1 -24980.809,E2 -24980.809} C_VEL
LIN {X 0,Y 180.994,Z 852.102,A -85,B 0,C 180,E1 -24981.542,E2 -24981.542} C_VEL
LIN {X 0,Y 181.42,Z 845.082,A -85,B 0,C 180,E1 -24981.961,E2 -24981.961} C_VEL
LIN {X 0,Y 181.721,Z 821.263,A -85,B 0,C 180,E1 -24983.797,E2 -24983.797} C_VEL
LIN {X 0,Y 181.687,Z 815.51,A -85,B 0,C 180,E1 -24984.33,E2 -24984.33} C_VEL
LIN {X 0,Y 178.991,Z 806.877,A -85,B 0,C 180,E1 -24986.866,E2 -24986.866} C_VEL
LIN {X 0,Y 176.73,Z 800.572,A -85,B 0,C 180,E1 -24989.182,E2 -24989.182} C_VEL
LIN {X 0,Y 174.835,Z 795.553,A -85,B 0,C 180,E1 -24991.397,E2 -24991.397} C_VEL
LIN {X 0,Y 173.09,Z 791.033,A -85,B 0,C 180,E1 -24993.718,E2 -24993.718} C_VEL
LIN {X 0,Y 170.566,Z 784.602,A -85,B 0,C 180,E1 -24998.077,E2 -24998.077} C_VEL
LIN {X 0,Y 168.644,Z 779.589,A -85,B 0,C 180,E1 -25003.663,E2 -25003.663} C_VEL
LIN {X 0,Y 168.287,Z 777.788,A -85,B 0,C 180,E1 -25006.749,E2 -25006.749} C_VEL
LIN {X 0,Y 168.481,Z 777.667,A -85,B 0,C 180,E1 -25011.674,E2 -25011.674} C_VEL
LIN {X 0,Y 170.156,Z 778.937,A -85,B 0,C 180,E1 -25017.041,E2 -25017.041} C_VEL
LIN {X 0,Y 171.684,Z 782.143,A -85,B 0,C 180,E1 -25020.272,E2 -25020.272} C_VEL
LIN {X 0,Y 172.952,Z 783.746,A -85,B 0,C 180,E1 -25022.161,E2 -25022.161} C_VEL
LIN {X 0,Y 175.249,Z 787.766,A -85,B 0,C 180,E1 -25025.178,E2 -25025.178} C_VEL
LIN {X 0,Y 178.022,Z 792.538,A -85,B 0,C 180,E1 -25028.112,E2 -25028.112} C_VEL
LIN {X 0,Y 181.238,Z 798.53,A -85,B 0,C 180,E1 -25031.006,E2 -25031.006} C_VEL
LIN {X 0,Y 184.717,Z 805.619,A -85,B 0,C 180,E1 -25033.75,E2 -25033.75} C_VEL
LIN {X 0,Y 185.093,Z 806.469,A -85,B 0,C 180,E1 -25034.028,E2 -25034.028} C_VEL
LIN {X 0,Y 183.426,Z 828.568,A -85,B 0,C 180,E1 -25035.119,E2 -25035.119} C_VEL
LIN {X 0,Y 181.524,Z 841.614,A -85,B 0,C 180,E1 -25036.139,E2 -25036.139} C_VEL
LIN {X 0,Y 178.974,Z 852.913,A -85,B 0,C 180,E1 -25037.323,E2 -25037.323} C_VEL
LIN {X 0,Y 175.729,Z 863.624,A -85,B 0,C 180,E1 -25038.777,E2 -25038.777} C_VEL
LIN {X 0,Y 171.282,Z 875.183,A -85,B 0,C 180,E1 -25040.834,E2 -25040.834} C_VEL
LIN {X 0,Y 166.325,Z 885.614,A -85,B 0,C 180,E1 -25043.225,E2 -25043.225} C_VEL
LIN {X 0,Y 160.85,Z 895.171,A -85,B 0,C 180,E1 -25046.121,E2 -25046.121} C_VEL
LIN {X 0,Y 155.36,Z 903.473,A -85,B 0,C 180,E1 -25049.459,E2 -25049.459} C_VEL
LIN {X 0,Y 150.46,Z 909.834,A -85,B 0,C 180,E1 -25052.785,E2 -25052.785} C_VEL
LIN {X 0,Y 145.305,Z 915.771,A -85,B 0,C 180,E1 -25057.062,E2 -25057.062} C_VEL
LIN {X 0,Y 140.785,Z 920.2,A -85,B 0,C 180,E1 -25061.52,E2 -25061.52} C_VEL
LIN {X 0,Y 137.306,Z 923.089,A -85,B 0,C 180,E1 -25065.775,E2 -25065.775} C_VEL
LIN {X 0,Y 134.121,Z 925.223,A -85,B 0,C 180,E1 -25071.044,E2 -25071.044} C_VEL
LIN {X 0,Y 132.645,Z 925.858,A -85,B 0,C 180,E1 -25074.357,E2 -25074.357} C_VEL
LIN {X 0,Y 131.188,Z 925.972,A -85,B 0,C 180,E1 -25079,E2 -25079} C_VEL
LIN {X 0,Y 130.342,Z 924.953,A -85,B 0,C 180,E1 -25084.452,E2 -25084.452} C_VEL
LIN {X 0,Y 130.287,Z 923.728,A -85,B 0,C 180,E1 -25087.82,E2 -25087.82} C_VEL
LIN {X 0,Y 130.909,Z 920.995,A -85,B 0,C 180,E1 -25092.831,E2 -25092.831} C_VEL
LIN {X 0,Y 132.263,Z 917.165,A -85,B 0,C 180,E1 -25097.733,E2 -25097.733} C_VEL
LIN {X 0,Y 134.562,Z 911.575,A -85,B 0,C 180,E1 -25102.914,E2 -25102.914} C_VEL
LIN {X 0,Y 137.502,Z 904.532,A -85,B 0,C 180,E1 -25107.807,E2 -25107.807} C_VEL
LIN {X 0,Y 140.638,Z 896.894,A -85,B 0,C 180,E1 -25111.881,E2 -25111.881} C_VEL
LIN {X 0,Y 144.087,Z 887.883,A -85,B 0,C 180,E1 -25115.602,E2 -25115.602} C_VEL
LIN {X 0,Y 147.627,Z 877.647,A -85,B 0,C 180,E1 -25118.905,E2 -25118.905} C_VEL
LIN {X 0,Y 150.529,Z 868.044,A -85,B 0,C 180,E1 -25121.341,E2 -25121.341} C_VEL
LIN {X 0,Y 153.497,Z 856.675,A -85,B 0,C 180,E1 -25123.575,E2 -25123.575} C_VEL
LIN {X 0,Y 156.086,Z 843.724,A -85,B 0,C 180,E1 -25125.51,E2 -25125.51} C_VEL
LIN {X 0,Y 157.885,Z 830.857,A -85,B 0,C 180,E1 -25126.901,E2 -25126.901} C_VEL
LIN {X 0,Y 158.943,Z 817.3,A -85,B 0,C 180,E1 -25127.872,E2 -25127.872} C_VEL
LIN {X 0,Y 160.16,Z 788.709,A -85,B 0,C 180,E1 -25129.268,E2 -25129.268} C_VEL
LIN {X 0,Y 155.9,Z 779.445,A -85,B 0,C 180,E1 -25131.115,E2 -25131.115} C_VEL
LIN {X 0,Y 148.245,Z 765.464,A -85,B 0,C 180,E1 -25134.604,E2 -25134.604} C_VEL
LIN {X 0,Y 140.978,Z 753.908,A -85,B 0,C 180,E1 -25138.334,E2 -25138.334} C_VEL
LIN {X 0,Y 137.966,Z 749.678,A -85,B 0,C 180,E1 -25140.003,E2 -25140.003} C_VEL
LIN {X 0,Y 135.314,Z 745.889,A -85,B 0,C 180,E1 -25141.574,E2 -25141.574} C_VEL
LIN {X 0,Y 133.068,Z 742.762,A -85,B 0,C 180,E1 -25142.976,E2 -25142.976} C_VEL
LIN {X 0,Y 132.392,Z 741.548,A -85,B 0,C 180,E1 -25143.44,E2 -25143.44} C_VEL
LIN {X 0,Y 130.089,Z 739.381,A -85,B 0,C 180,E1 -25144.91,E2 -25144.91} C_VEL
LIN {X 0,Y 129.097,Z 737.21,A -85,B 0,C 180,E1 -25145.875,E2 -25145.875} C_VEL
LIN {X 0,Y 128.935,Z 736.467,A -85,B 0,C 180,E1 -25146.846,E2 -25146.846} C_VEL
LIN {X 0,Y 129.08,Z 736.64,A -85,B 0,C 180,E1 -25150.669,E2 -25150.669} C_VEL
LIN {X 0,Y 129.281,Z 737.531,A -85,B 0,C 180,E1 -25151.111,E2 -25151.111} C_VEL
LIN {X 0,Y 140.115,Z 770.734,A -85,B 0,C 180,E1 -25155.26,E2 -25155.26} C_VEL
LIN {X 0,Y 137.453,Z 819.442,A -85,B 0,C 180,E1 -25159.354,E2 -25159.354} C_VEL
LIN {X 0,Y 136.475,Z 830.782,A -85,B 0,C 180,E1 -25160.695,E2 -25160.695} C_VEL
LIN {X 0,Y 135.386,Z 841.88,A -85,B 0,C 180,E1 -25162.413,E2 -25162.413} C_VEL
LIN {X 0,Y 134.21,Z 851.916,A -85,B 0,C 180,E1 -25164.368,E2 -25164.368} C_VEL
LIN {X 0,Y 133.018,Z 861.961,A -85,B 0,C 180,E1 -25166.758,E2 -25166.758} C_VEL
LIN {X 0,Y 131.927,Z 870.151,A -85,B 0,C 180,E1 -25169.072,E2 -25169.072} C_VEL
LIN {X 0,Y 130.828,Z 878.85,A -85,B 0,C 180,E1 -25171.962,E2 -25171.962} C_VEL
LIN {X 0,Y 129.961,Z 887.363,A -85,B 0,C 180,E1 -25175.303,E2 -25175.303} C_VEL
LIN {X 0,Y 129.355,Z 894.335,A -85,B 0,C 180,E1 -25178.485,E2 -25178.485} C_VEL
LIN {X 0,Y 129.022,Z 901.843,A -85,B 0,C 180,E1 -25182.566,E2 -25182.566} C_VEL
LIN {X 0,Y 129.152,Z 908.19,A -85,B 0,C 180,E1 -25186.628,E2 -25186.628} C_VEL
LIN {X 0,Y 129.868,Z 913.596,A -85,B 0,C 180,E1 -25190.656,E2 -25190.656} C_VEL
LIN {X 0,Y 131.462,Z 918.877,A -85,B 0,C 180,E1 -25195.4,E2 -25195.4} C_VEL
LIN {X 0,Y 133.891,Z 923.079,A -85,B 0,C 180,E1 -25200,E2 -25200} C_VEL
LIN {X 0,Y 135.9,Z 925.364,A -85,B 0,C 180,E1 -25202.964,E2 -25202.964} C_VEL
LIN {X 0,Y 141.063,Z 928.613,A -85,B 0,C 180,E1 -25208.596,E2 -25208.596} C_VEL
LIN {X 0,Y 144.079,Z 929.635,A -85,B 0,C 180,E1 -25211.251,E2 -25211.251} C_VEL
LIN {X 0,Y 151.15,Z 930.514,A -85,B 0,C 180,E1 -25216.199,E2 -25216.199} C_VEL
LIN {X 0,Y 159.249,Z 929.727,A -85,B 0,C 180,E1 -25220.674,E2 -25220.674} C_VEL
LIN {X 0,Y 163.746,Z 928.827,A -85,B 0,C 180,E1 -25222.723,E2 -25222.723} C_VEL
LIN {X 0,Y 173.183,Z 925.647,A -85,B 0,C 180,E1 -25226.512,E2 -25226.512} C_VEL
LIN {X 0,Y 180.782,Z 922.164,A -85,B 0,C 180,E1 -25229.074,E2 -25229.074} C_VEL
LIN {X 0,Y 188.76,Z 917.559,A -85,B 0,C 180,E1 -25231.416,E2 -25231.416} C_VEL
LIN {X 0,Y 195.68,Z 912.856,A -85,B 0,C 180,E1 -25233.21,E2 -25233.21} C_VEL
LIN {X 0,Y 204.471,Z 905.659,A -85,B 0,C 180,E1 -25235.281,E2 -25235.281} C_VEL
LIN {X 0,Y 203.368,Z 907.02,A -85,B 0,C 180,E1 -25235.807,E2 -25235.807} C_VEL
LIN {X 0,Y 194.229,Z 915.879,A -85,B 0,C 180,E1 -25237.241,E2 -25237.241} C_VEL
LIN {X 0,Y 182.451,Z 925.82,A -85,B 0,C 180,E1 -25239.606,E2 -25239.606} C_VEL
LIN {X 0,Y 174.063,Z 931.985,A -85,B 0,C 180,E1 -25241.667,E2 -25241.667} C_VEL
LIN {X 0,Y 166.09,Z 937.186,A -85,B 0,C 180,E1 -25243.995,E2 -25243.995} C_VEL
LIN {X 0,Y 156.408,Z 942.709,A -85,B 0,C 180,E1 -25247.618,E2 -25247.618} C_VEL
LIN {X 0,Y 147.966,Z 946.892,A -85,B 0,C 180,E1 -25251.864,E2 -25251.864} C_VEL
LIN {X 0,Y 140.776,Z 949.917,A -85,B 0,C 180,E1 -25256.686,E2 -25256.686} C_VEL
LIN {X 0,Y 135.124,Z 951.708,A -85,B 0,C 180,E1 -25262.152,E2 -25262.152} C_VEL
LIN {X 0,Y 133.067,Z 952.147,A -85,B 0,C 180,E1 -25265.001,E2 -25265.001} C_VEL
LIN {X 0,Y 130.503,Z 952.16,A -85,B 0,C 180,E1 -25270.262,E2 -25270.262} C_VEL
LIN {X 0,Y 129.032,Z 952.507,A -85,B 0,C 180,E1 -25272.767,E2 -25272.767} C_VEL
LIN {X 0,Y 126.866,Z 953.442,A -85,B 0,C 180,E1 -25275.2,E2 -25275.2} C_VEL
LIN {X 0,Y 122.537,Z 956.23,A -85,B 0,C 180,E1 -25280.17,E2 -25280.17} C_VEL
LIN {X 0,Y 121.449,Z 957.691,A -85,B 0,C 180,E1 -25282.839,E2 -25282.839} C_VEL
LIN {X 0,Y 121.393,Z 958.131,A -85,B 0,C 180,E1 -25283.754,E2 -25283.754} C_VEL
LIN {X 0,Y 121.666,Z 959.495,A -85,B 0,C 180,E1 -25286.684,E2 -25286.684} C_VEL
LIN {X 0,Y 122.164,Z 960.562,A -85,B 0,C 180,E1 -25289.995,E2 -25289.995} C_VEL
LIN {X 0,Y 121.558,Z 960.982,A -85,B 0,C 180,E1 -25293.309,E2 -25293.309} C_VEL
LIN {X 0,Y 120.905,Z 960.767,A -85,B 0,C 180,E1 -25298.821,E2 -25298.821} C_VEL
LIN {X 0,Y 121.021,Z 959.804,A -85,B 0,C 180,E1 -25303.427,E2 -25303.427} C_VEL
LIN {X 0,Y 122.655,Z 957.055,A -85,B 0,C 180,E1 -25310.103,E2 -25310.103} C_VEL
LIN {X 0,Y 125.076,Z 953.985,A -85,B 0,C 180,E1 -25314.919,E2 -25314.919} C_VEL
LIN {X 0,Y 128.642,Z 949.98,A -85,B 0,C 180,E1 -25319.446,E2 -25319.446} C_VEL
LIN {X 0,Y 132.895,Z 944.902,A -85,B 0,C 180,E1 -25323.724,E2 -25323.724} C_VEL
LIN {X 0,Y 139.014,Z 937.493,A -85,B 0,C 180,E1 -25328.26,E2 -25328.26} C_VEL
LIN {X 0,Y 145.001,Z 929.622,A -85,B 0,C 180,E1 -25331.787,E2 -25331.787} C_VEL
LIN {X 0,Y 150.554,Z 921.685,A -85,B 0,C 180,E1 -25334.438,E2 -25334.438} C_VEL
LIN {X 0,Y 157.062,Z 911.026,A -85,B 0,C 180,E1 -25337.109,E2 -25337.109} C_VEL
LIN {X 0,Y 162.682,Z 900.292,A -85,B 0,C 180,E1 -25339.108,E2 -25339.108} C_VEL
LIN {X 0,Y 167.168,Z 890.026,A -85,B 0,C 180,E1 -25340.574,E2 -25340.574} C_VEL
LIN {X 0,Y 171.805,Z 877.053,A -85,B 0,C 180,E1 -25341.902,E2 -25341.902} C_VEL
LIN {X 0,Y 175.371,Z 863.415,A -85,B 0,C 180,E1 -25342.905,E2 -25342.905} C_VEL
LIN {X 0,Y 177.618,Z 849.974,A -85,B 0,C 180,E1 -25343.593,E2 -25343.593} C_VEL
LIN {X 0,Y 178.303,Z 827.51,A -85,B 0,C 180,E1 -25345.31,E2 -25345.31} C_VEL
LIN {X 0,Y 178.311,Z 818.678,A -85,B 0,C 180,E1 -25346.155,E2 -25346.155} C_VEL
LIN {X 0,Y 175.831,Z 810.405,A -85,B 0,C 180,E1 -25348.773,E2 -25348.773} C_VEL
LIN {X 0,Y 173.371,Z 802.88,A -85,B 0,C 180,E1 -25351.788,E2 -25351.788} C_VEL
LIN {X 0,Y 171.299,Z 797.145,A -85,B 0,C 180,E1 -25354.788,E2 -25354.788} C_VEL
LIN {X 0,Y 169.154,Z 791.109,A -85,B 0,C 180,E1 -25358.926,E2 -25358.926} C_VEL
LIN {X 0,Y 167.534,Z 786.245,A -85,B 0,C 180,E1 -25364.489,E2 -25364.489} C_VEL
LIN {X 0,Y 167.315,Z 784.759,A -85,B 0,C 180,E1 -25367.107,E2 -25367.107} C_VEL
LIN {X 0,Y 167.526,Z 784.71,A -85,B 0,C 180,E1 -25371.626,E2 -25371.626} C_VEL
LIN {X 0,Y 168.969,Z 785.849,A -85,B 0,C 180,E1 -25376.537,E2 -25376.537} C_VEL
LIN {X 0,Y 170.522,Z 789.148,A -85,B 0,C 180,E1 -25380,E2 -25380} C_VEL
LIN {X 0,Y 171.58,Z 790.687,A -85,B 0,C 180,E1 -25381.668,E2 -25381.668} C_VEL
LIN {X 0,Y 173.573,Z 794.34,A -85,B 0,C 180,E1 -25384.467,E2 -25384.467} C_VEL
LIN {X 0,Y 176.686,Z 799.972,A -85,B 0,C 180,E1 -25387.906,E2 -25387.906} C_VEL
LIN {X 0,Y 180.535,Z 807.874,A -85,B 0,C 180,E1 -25391.448,E2 -25391.448} C_VEL
LIN {X 0,Y 181.456,Z 810.139,A -85,B 0,C 180,E1 -25392.235,E2 -25392.235} C_VEL
LIN {X 0,Y 179.823,Z 829.838,A -85,B 0,C 180,E1 -25393.23,E2 -25393.23} C_VEL
LIN {X 0,Y 177.846,Z 842.574,A -85,B 0,C 180,E1 -25394.233,E2 -25394.233} C_VEL
LIN {X 0,Y 175.012,Z 854.439,A -85,B 0,C 180,E1 -25395.483,E2 -25395.483} C_VEL
LIN {X 0,Y 171.198,Z 866.119,A -85,B 0,C 180,E1 -25397.107,E2 -25397.107} C_VEL
LIN {X 0,Y 166.491,Z 877.552,A -85,B 0,C 180,E1 -25399.194,E2 -25399.194} C_VEL
LIN {X 0,Y 161.476,Z 887.411,A -85,B 0,C 180,E1 -25401.527,E2 -25401.527} C_VEL
LIN {X 0,Y 155.686,Z 896.915,A -85,B 0,C 180,E1 -25404.477,E2 -25404.477} C_VEL
LIN {X 0,Y 150.506,Z 904.271,A -85,B 0,C 180,E1 -25407.483,E2 -25407.483} C_VEL
LIN {X 0,Y 145.303,Z 910.662,A -85,B 0,C 180,E1 -25410.858,E2 -25410.858} C_VEL
LIN {X 0,Y 140.651,Z 915.767,A -85,B 0,C 180,E1 -25414.474,E2 -25414.474} C_VEL
LIN {X 0,Y 135.669,Z 920.482,A -85,B 0,C 180,E1 -25419.018,E2 -25419.018} C_VEL
LIN {X 0,Y 131.247,Z 923.986,A -85,B 0,C 180,E1 -25424.118,E2 -25424.118} C_VEL
LIN {X 0,Y 127.135,Z 926.457,A -85,B 0,C 180,E1 -25430.708,E2 -25430.708} C_VEL
LIN {X 0,Y 125.022,Z 927.066,A -85,B 0,C 180,E1 -25435.802,E2 -25435.802} C_VEL
LIN {X 0,Y 124.045,Z 926.894,A -85,B 0,C 180,E1 -25439.348,E2 -25439.348} C_VEL
LIN {X 0,Y 123.444,Z 926.29,A -85,B 0,C 180,E1 -25442.911,E2 -25442.911} C_VEL
LIN {X 0,Y 123.255,Z 925.177,A -85,B 0,C 180,E1 -25446.481,E2 -25446.481} C_VEL
LIN {X 0,Y 123.647,Z 922.663,A -85,B 0,C 180,E1 -25451.788,E2 -25451.788} C_VEL
LIN {X 0,Y 124.922,Z 919.043,A -85,B 0,C 180,E1 -25457,E2 -25457} C_VEL
LIN {X 0,Y 126.854,Z 914.378,A -85,B 0,C 180,E1 -25461.942,E2 -25461.942} C_VEL
LIN {X 0,Y 129.525,Z 908.218,A -85,B 0,C 180,E1 -25466.894,E2 -25466.894} C_VEL
LIN {X 0,Y 132.808,Z 900.748,A -85,B 0,C 180,E1 -25471.446,E2 -25471.446} C_VEL
LIN {X 0,Y 136.136,Z 892.845,A -85,B 0,C 180,E1 -25475.188,E2 -25475.188} C_VEL
LIN {X 0,Y 140.086,Z 882.475,A -85,B 0,C 180,E1 -25479.024,E2 -25479.024} C_VEL
LIN {X 0,Y 143.331,Z 872.795,A -85,B 0,C 180,E1 -25481.79,E2 -25481.79} C_VEL
LIN {X 0,Y 146.494,Z 861.808,A -85,B 0,C 180,E1 -25484.237,E2 -25484.237} C_VEL
LIN {X 0,Y 149.453,Z 849.126,A -85,B 0,C 180,E1 -25486.393,E2 -25486.393} C_VEL
LIN {X 0,Y 151.609,Z 836.346,A -85,B 0,C 180,E1 -25487.973,E2 -25487.973} C_VEL
LIN {X 0,Y 152.946,Z 822.973,A -85,B 0,C 180,E1 -25489.15,E2 -25489.15} C_VEL
LIN {X 0,Y 154.586,Z 790.886,A -85,B 0,C 180,E1 -25490.793,E2 -25490.793} C_VEL
LIN {X 0,Y 149.622,Z 780.619,A -85,B 0,C 180,E1 -25493.073,E2 -25493.073} C_VEL
LIN {X 0,Y 143.005,Z 768.485,A -85,B 0,C 180,E1 -25496.381,E2 -25496.381} C_VEL
LIN {X 0,Y 136.489,Z 758.107,A -85,B 0,C 180,E1 -25499.985,E2 -25499.985} C_VEL
LIN {X 0,Y 131.452,Z 750.942,A -85,B 0,C 180,E1 -25503.097,E2 -25503.097} C_VEL
LIN {X 0,Y 129.061,Z 747.359,A -85,B 0,C 180,E1 -25504.743,E2 -25504.743} C_VEL
LIN {X 0,Y 126.483,Z 744.283,A -85,B 0,C 180,E1 -25506.585,E2 -25506.585} C_VEL
LIN {X 0,Y 125.718,Z 742.804,A -85,B 0,C 180,E1 -25507.22,E2 -25507.22} C_VEL
LIN {X 0,Y 123.359,Z 740.876,A -85,B 0,C 180,E1 -25509.006,E2 -25509.006} C_VEL
LIN {X 0,Y 122.764,Z 739.892,A -85,B 0,C 180,E1 -25509.785,E2 -25509.785} C_VEL
LIN {X 0,Y 122.947,Z 740.234,A -85,B 0,C 180,E1 -25510.36,E2 -25510.36} C_VEL
LIN {X 0,Y 123.736,Z 743.133,A -85,B 0,C 180,E1 -25511.008,E2 -25511.008} C_VEL
LIN {X 0,Y 133.082,Z 772.225,A -85,B 0,C 180,E1 -25514.757,E2 -25514.757} C_VEL
LIN {X 0,Y 130.424,Z 819.553,A -85,B 0,C 180,E1 -25518.98,E2 -25518.98} C_VEL
LIN {X 0,Y 129.298,Z 832.123,A -85,B 0,C 180,E1 -25520.559,E2 -25520.559} C_VEL
LIN {X 0,Y 128.154,Z 843.234,A -85,B 0,C 180,E1 -25522.403,E2 -25522.403} C_VEL
LIN {X 0,Y 126.983,Z 853.219,A -85,B 0,C 180,E1 -25524.469,E2 -25524.469} C_VEL
LIN {X 0,Y 125.738,Z 863.192,A -85,B 0,C 180,E1 -25526.981,E2 -25526.981} C_VEL
LIN {X 0,Y 124.475,Z 872.885,A -85,B 0,C 180,E1 -25529.927,E2 -25529.927} C_VEL
LIN {X 0,Y 123.472,Z 881.108,A -85,B 0,C 180,E1 -25532.911,E2 -25532.911} C_VEL
LIN {X 0,Y 122.651,Z 889.164,A -85,B 0,C 180,E1 -25536.352,E2 -25536.352} C_VEL
LIN {X 0,Y 122.165,Z 896.133,A -85,B 0,C 180,E1 -25539.807,E2 -25539.807} C_VEL
LIN {X 0,Y 121.95,Z 903.542,A -85,B 0,C 180,E1 -25544.112,E2 -25544.112} C_VEL
LIN {X 0,Y 122.21,Z 909.131,A -85,B 0,C 180,E1 -25547.879,E2 -25547.879} C_VEL
LIN {X 0,Y 123.026,Z 914.178,A -85,B 0,C 180,E1 -25551.789,E2 -25551.789} C_VEL
LIN {X 0,Y 124.867,Z 919.615,A -85,B 0,C 180,E1 -25556.773,E2 -25556.773} C_VEL
LIN {X 0,Y 127.533,Z 923.953,A -85,B 0,C 180,E1 -25561.578,E2 -25561.578} C_VEL
LIN {X 0,Y 131.044,Z 927.311,A -85,B 0,C 180,E1 -25566.157,E2 -25566.157} C_VEL
LIN {X 0,Y 136.941,Z 930.338,A -85,B 0,C 180,E1 -25571.846,E2 -25571.846} C_VEL
LIN {X 0,Y 140.448,Z 931.283,A -85,B 0,C 180,E1 -25574.489,E2 -25574.489} C_VEL
LIN {X 0,Y 144.235,Z 931.82,A -85,B 0,C 180,E1 -25576.999,E2 -25576.999} C_VEL
LIN {X 0,Y 152.621,Z 931.684,A -85,B 0,C 180,E1 -25581.616,E2 -25581.616} C_VEL
LIN {X 0,Y 162.035,Z 930.05,A -85,B 0,C 180,E1 -25585.704,E2 -25585.704} C_VEL
LIN {X 0,Y 172.158,Z 926.701,A -85,B 0,C 180,E1 -25589.332,E2 -25589.332} C_VEL
LIN {X 0,Y 180.261,Z 923.089,A -85,B 0,C 180,E1 -25591.758,E2 -25591.758} C_VEL
LIN {X 0,Y 188.742,Z 918.324,A -85,B 0,C 180,E1 -25593.955,E2 -25593.955} C_VEL
LIN {X 0,Y 191.979,Z 916.335,A -85,B 0,C 180,E1 -25594.726,E2 -25594.726} C_VEL
LIN {X 0,Y 191.573,Z 916.916,A -85,B 0,C 180,E1 -25595.318,E2 -25595.318} C_VEL
LIN {X 0,Y 180.994,Z 925.089,A -85,B 0,C 180,E1 -25597.244,E2 -25597.244} C_VEL
LIN {X 0,Y 172.268,Z 931.071,A -85,B 0,C 180,E1 -25599.177,E2 -25599.177} C_VEL
LIN {X 0,Y 163.947,Z 936.113,A -85,B 0,C 180,E1 -25601.389,E2 -25601.389} C_VEL
LIN {X 0,Y 156.137,Z 940.33,A -85,B 0,C 180,E1 -25603.925,E2 -25603.925} C_VEL
LIN {X 0,Y 146.668,Z 944.689,A -85,B 0,C 180,E1 -25607.862,E2 -25607.862} C_VEL
LIN {X 0,Y 138.536,Z 947.851,A -85,B 0,C 180,E1 -25612.495,E2 -25612.495} C_VEL
LIN {X 0,Y 131.758,Z 949.827,A -85,B 0,C 180,E1 -25617.759,E2 -25617.759} C_VEL
LIN {X 0,Y 126.725,Z 950.597,A -85,B 0,C 180,E1 -25623.657,E2 -25623.657} C_VEL
LIN {X 0,Y 123.764,Z 950.318,A -85,B 0,C 180,E1 -25629.766,E2 -25629.766} C_VEL
LIN {X 0,Y 122.918,Z 950.059,A -85,B 0,C 180,E1 -25632.849,E2 -25632.849} C_VEL
LIN {X 0,Y 121.482,Z 954.756,A -85,B 0,C 180,E1 -25638.313,E2 -25638.313} C_VEL
LIN {X 0,Y 121.393,Z 958.131,A -85,B 0,C 180,E1 -25643.754,E2 -25643.754} C_VEL
LIN {X 0,Y 121.123,Z 958.95,A -85,B 0,C 180,E1 -25645.575,E2 -25645.575} C_VEL
LIN {X 0,Y 119.775,Z 959.738,A -85,B 0,C 180,E1 -25648.3,E2 -25648.3} C_VEL
LIN {X 0,Y 116.459,Z 960.16,A -85,B 0,C 180,E1 -25652.909,E2 -25652.909} C_VEL
LIN {X 0,Y 114.298,Z 959.983,A -85,B 0,C 180,E1 -25656.822,E2 -25656.822} C_VEL
LIN {X 0,Y 113.862,Z 959.814,A -85,B 0,C 180,E1 -25658.855,E2 -25658.855} C_VEL
LIN {X 0,Y 114.055,Z 958.841,A -85,B 0,C 180,E1 -25664.264,E2 -25664.264} C_VEL
LIN {X 0,Y 114.782,Z 957.729,A -85,B 0,C 180,E1 -25667.822,E2 -25667.822} C_VEL
LIN {X 0,Y 117.587,Z 954.307,A -85,B 0,C 180,E1 -25674.726,E2 -25674.726} C_VEL
LIN {X 0,Y 120.643,Z 951.125,A -85,B 0,C 180,E1 -25679.096,E2 -25679.096} C_VEL
LIN {X 0,Y 125.417,Z 946.124,A -85,B 0,C 180,E1 -25684.075,E2 -25684.075} C_VEL
LIN {X 0,Y 130.568,Z 940.414,A -85,B 0,C 180,E1 -25688.237,E2 -25688.237} C_VEL
LIN {X 0,Y 136.528,Z 933.419,A -85,B 0,C 180,E1 -25691.999,E2 -25691.999} C_VEL
LIN {X 0,Y 143.188,Z 924.879,A -85,B 0,C 180,E1 -25695.367,E2 -25695.367} C_VEL
LIN {X 0,Y 149.226,Z 916.22,A -85,B 0,C 180,E1 -25697.876,E2 -25697.876} C_VEL
LIN {X 0,Y 155.493,Z 905.667,A -85,B 0,C 180,E1 -25700.201,E2 -25700.201} C_VEL
LIN {X 0,Y 160.778,Z 895.351,A -85,B 0,C 180,E1 -25701.883,E2 -25701.883} C_VEL
LIN {X 0,Y 165.544,Z 884.179,A -85,B 0,C 180,E1 -25703.249,E2 -25703.249} C_VEL
LIN {X 0,Y 169.822,Z 871.283,A -85,B 0,C 180,E1 -25704.421,E2 -25704.421} C_VEL
LIN {X 0,Y 173.163,Z 857.195,A -85,B 0,C 180,E1 -25705.287,E2 -25705.287} C_VEL
LIN {X 0,Y 174.282,Z 849.878,A -85,B 0,C 180,E1 -25705.672,E2 -25705.672} C_VEL
LIN {X 0,Y 175.121,Z 828.322,A -85,B 0,C 180,E1 -25707.366,E2 -25707.366} C_VEL
LIN {X 0,Y 175.176,Z 822.174,A -85,B 0,C 180,E1 -25707.976,E2 -25707.976} C_VEL
LIN {X 0,Y 173.074,Z 814.452,A -85,B 0,C 180,E1 -25710.572,E2 -25710.572} C_VEL
LIN {X 0,Y 170.853,Z 807.345,A -85,B 0,C 180,E1 -25713.674,E2 -25713.674} C_VEL
LIN {X 0,Y 169.531,Z 803.108,A -85,B 0,C 180,E1 -25715.956,E2 -25715.956} C_VEL
LIN {X 0,Y 167.78,Z 797.559,A -85,B 0,C 180,E1 -25719.851,E2 -25719.851} C_VEL
LIN {X 0,Y 166.486,Z 793.017,A -85,B 0,C 180,E1 -25725.148,E2 -25725.148} C_VEL
LIN {X 0,Y 166.366,Z 791.89,A -85,B 0,C 180,E1 -25727.032,E2 -25727.032} C_VEL
LIN {X 0,Y 166.572,Z 791.754,A -85,B 0,C 180,E1 -25731.578,E2 -25731.578} C_VEL
LIN {X 0,Y 167.786,Z 792.742,A -85,B 0,C 180,E1 -25736.002,E2 -25736.002} C_VEL
LIN {X 0,Y 169.292,Z 796.047,A -85,B 0,C 180,E1 -25739.598,E2 -25739.598} C_VEL
LIN {X 0,Y 170.106,Z 797.306,A -85,B 0,C 180,E1 -25740.96,E2 -25740.96} C_VEL
LIN {X 0,Y 171.975,Z 801.015,A -85,B 0,C 180,E1 -25743.775,E2 -25743.775} C_VEL
LIN {X 0,Y 174.439,Z 805.747,A -85,B 0,C 180,E1 -25746.738,E2 -25746.738} C_VEL
LIN {X 0,Y 177.987,Z 813.45,A -85,B 0,C 180,E1 -25750.318,E2 -25750.318} C_VEL
LIN {X 0,Y 176.393,Z 831.73,A -85,B 0,C 180,E1 -25751.312,E2 -25751.312} C_VEL
LIN {X 0,Y 174.218,Z 844.549,A -85,B 0,C 180,E1 -25752.327,E2 -25752.327} C_VEL
LIN {X 0,Y 171.132,Z 856.466,A -85,B 0,C 180,E1 -25753.608,E2 -25753.608} C_VEL
LIN {X 0,Y 167.42,Z 867.235,A -85,B 0,C 180,E1 -25755.11,E2 -25755.11} C_VEL
LIN {X 0,Y 162.674,Z 878.219,A -85,B 0,C 180,E1 -25757.1,E2 -25757.1} C_VEL
LIN {X 0,Y 157.925,Z 887.247,A -85,B 0,C 180,E1 -25759.188,E2 -25759.188} C_VEL
LIN {X 0,Y 151.766,Z 897.074,A -85,B 0,C 180,E1 -25762.168,E2 -25762.168} C_VEL
LIN {X 0,Y 145.732,Z 905.248,A -85,B 0,C 180,E1 -25765.468,E2 -25765.468} C_VEL
LIN {X 0,Y 140.328,Z 911.519,A -85,B 0,C 180,E1 -25768.793,E2 -25768.793} C_VEL
LIN {X 0,Y 134.423,Z 917.56,A -85,B 0,C 180,E1 -25773.234,E2 -25773.234} C_VEL
LIN {X 0,Y 129.194,Z 922.049,A -85,B 0,C 180,E1 -25777.936,E2 -25777.936} C_VEL
LIN {X 0,Y 124.775,Z 925.224,A -85,B 0,C 180,E1 -25782.934,E2 -25782.934} C_VEL
LIN {X 0,Y 122.323,Z 926.69,A -85,B 0,C 180,E1 -25786.42,E2 -25786.42} C_VEL
LIN {X 0,Y 120.299,Z 927.6,A -85,B 0,C 180,E1 -25790.019,E2 -25790.019} C_VEL
LIN {X 0,Y 117.643,Z 928.087,A -85,B 0,C 180,E1 -25796.759,E2 -25796.759} C_VEL
LIN {X 0,Y 116.642,Z 927.538,A -85,B 0,C 180,E1 -25801.189,E2 -25801.189} C_VEL
LIN {X 0,Y 116.224,Z 926.568,A -85,B 0,C 180,E1 -25805.102,E2 -25805.102} C_VEL
LIN {X 0,Y 116.263,Z 925.174,A -85,B 0,C 180,E1 -25808.74,E2 -25808.74} C_VEL
LIN {X 0,Y 117.022,Z 922.405,A -85,B 0,C 180,E1 -25813.931,E2 -25813.931} C_VEL
LIN {X 0,Y 118.734,Z 917.993,A -85,B 0,C 180,E1 -25819.777,E2 -25819.777} C_VEL
LIN {X 0,Y 121.187,Z 912.617,A -85,B 0,C 180,E1 -25825.015,E2 -25825.015} C_VEL
LIN {X 0,Y 124.316,Z 905.891,A -85,B 0,C 180,E1 -25830.005,E2 -25830.005} C_VEL
LIN {X 0,Y 128.089,Z 897.463,A -85,B 0,C 180,E1 -25834.726,E2 -25834.726} C_VEL
LIN {X 0,Y 131.705,Z 888.876,A -85,B 0,C 180,E1 -25838.443,E2 -25838.443} C_VEL
LIN {X 0,Y 135.672,Z 878.398,A -85,B 0,C 180,E1 -25841.963,E2 -25841.963} C_VEL
LIN {X 0,Y 139.444,Z 866.584,A -85,B 0,C 180,E1 -25844.974,E2 -25844.974} C_VEL
LIN {X 0,Y 142.588,Z 854.964,A -85,B 0,C 180,E1 -25847.206,E2 -25847.206} C_VEL
LIN {X 0,Y 145.214,Z 841.882,A -85,B 0,C 180,E1 -25849.072,E2 -25849.072} C_VEL
LIN {X 0,Y 147.005,Z 828.684,A -85,B 0,C 180,E1 -25850.418,E2 -25850.418} C_VEL
LIN {X 0,Y 147.957,Z 814.62,A -85,B 0,C 180,E1 -25851.336,E2 -25851.336} C_VEL
LIN {X 0,Y 149.018,Z 793.093,A -85,B 0,C 180,E1 -25852.432,E2 -25852.432} C_VEL
LIN {X 0,Y 143.17,Z 781.144,A -85,B 0,C 180,E1 -25855.374,E2 -25855.374} C_VEL
LIN {X 0,Y 137.315,Z 770.575,A -85,B 0,C 180,E1 -25858.588,E2 -25858.588} C_VEL
LIN {X 0,Y 131.392,Z 761.161,A -85,B 0,C 180,E1 -25862.219,E2 -25862.219} C_VEL
LIN {X 0,Y 125.739,Z 752.957,A -85,B 0,C 180,E1 -25866.172,E2 -25866.172} C_VEL
LIN {X 0,Y 123.103,Z 749.38,A -85,B 0,C 180,E1 -25868.242,E2 -25868.242} C_VEL
LIN {X 0,Y 122.871,Z 748.971,A -85,B 0,C 180,E1 -25868.445,E2 -25868.445} C_VEL
LIN {X 0,Y 122.132,Z 749.841,A -85,B 0,C 180,E1 -25868.857,E2 -25868.857} C_VEL
LIN {X 0,Y 120.936,Z 751.136,A -85,B 0,C 180,E1 -25869.548,E2 -25869.548} C_VEL
LIN {X 0,Y 119.662,Z 751.896,A -85,B 0,C 180,E1 -25870.691,E2 -25870.691} C_VEL
LIN {X 0,Y 119.843,Z 753.556,A -85,B 0,C 180,E1 -25871.486,E2 -25871.486} C_VEL
LIN {X 0,Y 122.98,Z 763.502,A -85,B 0,C 180,E1 -25872.976,E2 -25872.976} C_VEL
LIN {X 0,Y 126.031,Z 773.239,A -85,B 0,C 180,E1 -25874.232,E2 -25874.232} C_VEL
LIN {X 0,Y 123.237,Z 820.868,A -85,B 0,C 180,E1 -25878.746,E2 -25878.746} C_VEL
LIN {X 0,Y 122.228,Z 832.194,A -85,B 0,C 180,E1 -25880.231,E2 -25880.231} C_VEL
LIN {X 0,Y 121.037,Z 843.457,A -85,B 0,C 180,E1 -25882.17,E2 -25882.17} C_VEL
LIN {X 0,Y 119.808,Z 853.723,A -85,B 0,C 180,E1 -25884.398,E2 -25884.398} C_VEL
LIN {X 0,Y 118.534,Z 863.885,A -85,B 0,C 180,E1 -25887.117,E2 -25887.117} C_VEL
LIN {X 0,Y 117.378,Z 872.584,A -85,B 0,C 180,E1 -25889.903,E2 -25889.903} C_VEL
LIN {X 0,Y 116.239,Z 882.055,A -85,B 0,C 180,E1 -25893.518,E2 -25893.518} C_VEL
LIN {X 0,Y 115.459,Z 889.885,A -85,B 0,C 180,E1 -25897.041,E2 -25897.041} C_VEL
LIN {X 0,Y 115.072,Z 896.342,A -85,B 0,C 180,E1 -25900.371,E2 -25900.371} C_VEL
LIN {X 0,Y 114.9,Z 903.811,A -85,B 0,C 180,E1 -25904.932,E2 -25904.932} C_VEL
LIN {X 0,Y 115.584,Z 911.311,A -85,B 0,C 180,E1 -25910.374,E2 -25910.374} C_VEL
LIN {X 0,Y 116.83,Z 916.584,A -85,B 0,C 180,E1 -25914.822,E2 -25914.822} C_VEL
LIN {X 0,Y 119.233,Z 921.766,A -85,B 0,C 180,E1 -25919.999,E2 -25919.999} C_VEL
LIN {X 0,Y 122.467,Z 925.929,A -85,B 0,C 180,E1 -25924.938,E2 -25924.938} C_VEL
LIN {X 0,Y 126.631,Z 929.132,A -85,B 0,C 180,E1 -25929.584,E2 -25929.584} C_VEL
LIN {X 0,Y 133.399,Z 932.055,A -85,B 0,C 180,E1 -25935.273,E2 -25935.273} C_VEL
LIN {X 0,Y 141.521,Z 933.333,A -85,B 0,C 180,E1 -25940.342,E2 -25940.342} C_VEL
LIN {X 0,Y 150.746,Z 933.107,A -85,B 0,C 180,E1 -25944.809,E2 -25944.809} C_VEL
LIN {X 0,Y 160.849,Z 931.252,A -85,B 0,C 180,E1 -25948.726,E2 -25948.726} C_VEL
LIN {X 0,Y 166.164,Z 929.796,A -85,B 0,C 180,E1 -25950.5,E2 -25950.5} C_VEL
LIN {X 0,Y 177.467,Z 925.429,A -85,B 0,C 180,E1 -25953.727,E2 -25953.727} C_VEL
LIN {X 0,Y 179.882,Z 924.5,A -85,B 0,C 180,E1 -25954.863,E2 -25954.863} C_VEL
LIN {X 0,Y 170.829,Z 930.237,A -85,B 0,C 180,E1 -25956.65,E2 -25956.65} C_VEL
LIN {X 0,Y 162.118,Z 935.106,A -85,B 0,C 180,E1 -25958.705,E2 -25958.705} C_VEL
LIN {X 0,Y 153.949,Z 939.159,A -85,B 0,C 180,E1 -25961.122,E2 -25961.122} C_VEL
LIN {X 0,Y 146.252,Z 942.487,A -85,B 0,C 180,E1 -25963.873,E2 -25963.873} C_VEL
LIN {X 0,Y 137.096,Z 945.799,A -85,B 0,C 180,E1 -25968.203,E2 -25968.203} C_VEL
LIN {X 0,Y 129.211,Z 947.948,A -85,B 0,C 180,E1 -25973.246,E2 -25973.246} C_VEL
LIN {X 0,Y 122.788,Z 948.963,A -85,B 0,C 180,E1 -25979.154,E2 -25979.154} C_VEL
LIN {X 0,Y 118.539,Z 948.877,A -85,B 0,C 180,E1 -25985.474,E2 -25985.474} C_VEL
LIN {X 0,Y 116.422,Z 948.155,A -85,B 0,C 180,E1 -25991.29,E2 -25991.29} C_VEL
LIN {X 0,Y 114.537,Z 953.437,A -85,B 0,C 180,E1 -25997.593,E2 -25997.593} C_VEL
LIN {X 0,Y 114.364,Z 957.156,A -85,B 0,C 180,E1 -26003.935,E2 -26003.935} C_VEL
LIN {X 0,Y 114.596,Z 958.301,A -85,B 0,C 180,E1 -26006.479,E2 -26006.479} C_VEL
LIN {X 0,Y 115.101,Z 959.446,A -85,B 0,C 180,E1 -26009.995,E2 -26009.995} C_VEL
LIN {X 0,Y 114.477,Z 959.899,A -85,B 0,C 180,E1 -26013.514,E2 -26013.514} C_VEL
LIN {X 0,Y 113.862,Z 959.814,A -85,B 0,C 180,E1 -26018.855,E2 -26018.855} C_VEL
LIN {X 0,Y 113.168,Z 959.396,A -85,B 0,C 180,E1 -26021.81,E2 -26021.81} C_VEL
LIN {X 0,Y 110.94,Z 957.939,A -85,B 0,C 180,E1 -26026.698,E2 -26026.698} C_VEL
LIN {X 0,Y 109.659,Z 956.279,A -85,B 0,C 180,E1 -26030.689,E2 -26030.689} C_VEL
LIN {X 0,Y 109.854,Z 954.885,A -85,B 0,C 180,E1 -26033.689,E2 -26033.689} C_VEL
LIN {X 0,Y 110.25,Z 954.357,A -85,B 0,C 180,E1 -26034.663,E2 -26034.663} C_VEL
LIN {X 0,Y 114.109,Z 950.756,A -85,B 0,C 180,E1 -26040.429,E2 -26040.429} C_VEL
LIN {X 0,Y 119.555,Z 945.548,A -85,B 0,C 180,E1 -26045.998,E2 -26045.998} C_VEL
LIN {X 0,Y 126.06,Z 938.896,A -85,B 0,C 180,E1 -26050.919,E2 -26050.919} C_VEL
LIN {X 0,Y 132.444,Z 931.823,A -85,B 0,C 180,E1 -26054.669,E2 -26054.669} C_VEL
LIN {X 0,Y 139.533,Z 923.19,A -85,B 0,C 180,E1 -26057.974,E2 -26057.974} C_VEL
LIN {X 0,Y 145.795,Z 914.418,A -85,B 0,C 180,E1 -26060.462,E2 -26060.462} C_VEL
LIN {X 0,Y 152.453,Z 903.728,A -85,B 0,C 180,E1 -26062.668,E2 -26062.668} C_VEL
LIN {X 0,Y 157.868,Z 893.244,A -85,B 0,C 180,E1 -26064.33,E2 -26064.33} C_VEL
LIN {X 0,Y 162.751,Z 882.057,A -85,B 0,C 180,E1 -26065.595,E2 -26065.595} C_VEL
LIN {X 0,Y 167.05,Z 869.141,A -85,B 0,C 180,E1 -26066.689,E2 -26066.689} C_VEL
LIN {X 0,Y 170.351,Z 855.276,A -85,B 0,C 180,E1 -26067.503,E2 -26067.503} C_VEL
LIN {X 0,Y 171.247,Z 848.964,A -85,B 0,C 180,E1 -26067.886,E2 -26067.886} C_VEL
LIN {X 0,Y 172.334,Z 826.038,A -85,B 0,C 180,E1 -26069.787,E2 -26069.787} C_VEL
LIN {X 0,Y 170.768,Z 819.605,A -85,B 0,C 180,E1 -26072.011,E2 -26072.011} C_VEL
LIN {X 0,Y 168.928,Z 812.928,A -85,B 0,C 180,E1 -26075.006,E2 -26075.006} C_VEL
LIN {X 0,Y 167.874,Z 809.222,A -85,B 0,C 180,E1 -26077.066,E2 -26077.066} C_VEL
LIN {X 0,Y 166.455,Z 804.019,A -85,B 0,C 180,E1 -26080.778,E2 -26080.778} C_VEL
LIN {X 0,Y 165.469,Z 799.854,A -85,B 0,C 180,E1 -26085.71,E2 -26085.71} C_VEL
LIN {X 0,Y 165.387,Z 798.77,A -85,B 0,C 180,E1 -26087.767,E2 -26087.767} C_VEL
LIN {X 0,Y 165.618,Z 798.797,A -85,B 0,C 180,E1 -26091.529,E2 -26091.529} C_VEL
LIN {X 0,Y 166.679,Z 799.832,A -85,B 0,C 180,E1 -26095.668,E2 -26095.668} C_VEL
LIN {X 0,Y 168.317,Z 803.246,A -85,B 0,C 180,E1 -26099.616,E2 -26099.616} C_VEL
LIN {X 0,Y 170.255,Z 807.307,A -85,B 0,C 180,E1 -26102.843,E2 -26102.843} C_VEL
LIN {X 0,Y 172.679,Z 812.371,A -85,B 0,C 180,E1 -26106.027,E2 -26106.027} C_VEL
LIN {X 0,Y 174.808,Z 817.563,A -85,B 0,C 180,E1 -26108.433,E2 -26108.433} C_VEL
LIN {X 0,Y 173.264,Z 833.058,A -85,B 0,C 180,E1 -26109.271,E2 -26109.271} C_VEL
LIN {X 0,Y 170.953,Z 845.804,A -85,B 0,C 180,E1 -26110.279,E2 -26110.279} C_VEL
LIN {X 0,Y 167.666,Z 857.801,A -85,B 0,C 180,E1 -26111.561,E2 -26111.561} C_VEL
LIN {X 0,Y 163.333,Z 869.664,A -85,B 0,C 180,E1 -26113.232,E2 -26113.232} C_VEL
LIN {X 0,Y 158.265,Z 880.613,A -85,B 0,C 180,E1 -26115.254,E2 -26115.254} C_VEL
LIN {X 0,Y 152.91,Z 890.036,A -85,B 0,C 180,E1 -26117.519,E2 -26117.519} C_VEL
LIN {X 0,Y 146.366,Z 899.68,A -85,B 0,C 180,E1 -26120.57,E2 -26120.57} C_VEL
LIN {X 0,Y 140.768,Z 906.732,A -85,B 0,C 180,E1 -26123.542,E2 -26123.542} C_VEL
LIN {X 0,Y 134.449,Z 913.534,A -85,B 0,C 180,E1 -26127.309,E2 -26127.309} C_VEL
LIN {X 0,Y 128.251,Z 919.309,A -85,B 0,C 180,E1 -26131.865,E2 -26131.865} C_VEL
LIN {X 0,Y 122.771,Z 923.623,A -85,B 0,C 180,E1 -26136.742,E2 -26136.742} C_VEL
LIN {X 0,Y 119.442,Z 925.84,A -85,B 0,C 180,E1 -26140.335,E2 -26140.335} C_VEL
LIN {X 0,Y 116.774,Z 927.345,A -85,B 0,C 180,E1 -26143.77,E2 -26143.77} C_VEL
LIN {X 0,Y 114.431,Z 928.445,A -85,B 0,C 180,E1 -26147.508,E2 -26147.508} C_VEL
LIN {X 0,Y 112.485,Z 929.012,A -85,B 0,C 180,E1 -26151.34,E2 -26151.34} C_VEL
LIN {X 0,Y 110.955,Z 929.127,A -85,B 0,C 180,E1 -26155.432,E2 -26155.432} C_VEL
LIN {X 0,Y 109.945,Z 928.786,A -85,B 0,C 180,E1 -26159.251,E2 -26159.251} C_VEL
LIN {X 0,Y 109.243,Z 927.694,A -85,B 0,C 180,E1 -26164.249,E2 -26164.249} C_VEL
LIN {X 0,Y 109.466,Z 924.929,A -85,B 0,C 180,E1 -26171.282,E2 -26171.282} C_VEL
LIN {X 0,Y 110.726,Z 921.374,A -85,B 0,C 180,E1 -26177.17,E2 -26177.17} C_VEL
LIN {X 0,Y 113.17,Z 916,A -85,B 0,C 180,E1 -26183.533,E2 -26183.533} C_VEL
LIN {X 0,Y 116.254,Z 909.568,A -85,B 0,C 180,E1 -26189.139,E2 -26189.139} C_VEL
LIN {X 0,Y 120.099,Z 901.638,A -85,B 0,C 180,E1 -26194.279,E2 -26194.279} C_VEL
LIN {X 0,Y 123.699,Z 893.854,A -85,B 0,C 180,E1 -26198.171,E2 -26198.171} C_VEL
LIN {X 0,Y 127.702,Z 884.307,A -85,B 0,C 180,E1 -26201.915,E2 -26201.915} C_VEL
LIN {X 0,Y 131.556,Z 873.829,A -85,B 0,C 180,E1 -26205.055,E2 -26205.055} C_VEL
LIN {X 0,Y 135.269,Z 861.925,A -85,B 0,C 180,E1 -26207.777,E2 -26207.777} C_VEL
LIN {X 0,Y 138.296,Z 849.696,A -85,B 0,C 180,E1 -26209.872,E2 -26209.872} C_VEL
LIN {X 0,Y 140.706,Z 836.12,A -85,B 0,C 180,E1 -26211.556,E2 -26211.556} C_VEL
LIN {X 0,Y 142.072,Z 823.194,A -85,B 0,C 180,E1 -26212.675,E2 -26212.675} C_VEL
LIN {X 0,Y 143.661,Z 795.603,A -85,B 0,C 180,E1 -26214.135,E2 -26214.135} C_VEL
LIN {X 0,Y 136.893,Z 781.825,A -85,B 0,C 180,E1 -26217.869,E2 -26217.869} C_VEL
LIN {X 0,Y 131.671,Z 772.689,A -85,B 0,C 180,E1 -26221.052,E2 -26221.052} C_VEL
LIN {X 0,Y 127.235,Z 765.589,A -85,B 0,C 180,E1 -26224.049,E2 -26224.049} C_VEL
LIN {X 0,Y 122.61,Z 758.659,A -85,B 0,C 180,E1 -26227.563,E2 -26227.563} C_VEL
LIN {X 0,Y 121.689,Z 757.645,A -85,B 0,C 180,E1 -26228.293,E2 -26228.293} C_VEL
LIN {X 0,Y 120.965,Z 758.09,A -85,B 0,C 180,E1 -26228.744,E2 -26228.744} C_VEL
LIN {X 0,Y 119.236,Z 762.015,A -85,B 0,C 180,E1 -26229.519,E2 -26229.519} C_VEL
LIN {X 0,Y 117.886,Z 763.742,A -85,B 0,C 180,E1 -26230.304,E2 -26230.304} C_VEL
LIN {X 0,Y 116.407,Z 764.736,A -85,B 0,C 180,E1 -26231.621,E2 -26231.621} C_VEL
LIN {X 0,Y 116.574,Z 766.296,A -85,B 0,C 180,E1 -26232.421,E2 -26232.421} C_VEL
LIN {X 0,Y 119.008,Z 774.015,A -85,B 0,C 180,E1 -26233.632,E2 -26233.632} C_VEL
LIN {X 0,Y 116.173,Z 821.447,A -85,B 0,C 180,E1 -26238.427,E2 -26238.427} C_VEL
LIN {X 0,Y 115.041,Z 833.318,A -85,B 0,C 180,E1 -26240.098,E2 -26240.098} C_VEL
LIN {X 0,Y 113.944,Z 843.32,A -85,B 0,C 180,E1 -26241.917,E2 -26241.917} C_VEL
LIN {X 0,Y 112.634,Z 854.156,A -85,B 0,C 180,E1 -26244.389,E2 -26244.389} C_VEL
LIN {X 0,Y 111.42,Z 863.667,A -85,B 0,C 180,E1 -26247.04,E2 -26247.04} C_VEL
LIN {X 0,Y 110.092,Z 873.487,A -85,B 0,C 180,E1 -26250.347,E2 -26250.347} C_VEL
LIN {X 0,Y 109.137,Z 881.888,A -85,B 0,C 180,E1 -26253.72,E2 -26253.72} C_VEL
LIN {X 0,Y 108.303,Z 890.979,A -85,B 0,C 180,E1 -26258.091,E2 -26258.091} C_VEL
LIN {X 0,Y 107.932,Z 897.929,A -85,B 0,C 180,E1 -26261.982,E2 -26261.982} C_VEL
LIN {X 0,Y 108.048,Z 906.079,A -85,B 0,C 180,E1 -26267.362,E2 -26267.362} C_VEL
LIN {X 0,Y 108.974,Z 912.748,A -85,B 0,C 180,E1 -26272.588,E2 -26272.588} C_VEL
LIN {X 0,Y 110.215,Z 917.055,A -85,B 0,C 180,E1 -26276.343,E2 -26276.343} C_VEL
LIN {X 0,Y 113.196,Z 922.856,A -85,B 0,C 180,E1 -26282.307,E2 -26282.307} C_VEL
LIN {X 0,Y 116.448,Z 926.721,A -85,B 0,C 180,E1 -26286.932,E2 -26286.932} C_VEL
LIN {X 0,Y 122.782,Z 930.967,A -85,B 0,C 180,E1 -26293.306,E2 -26293.306} C_VEL
LIN {X 0,Y 126.377,Z 932.562,A -85,B 0,C 180,E1 -26296.144,E2 -26296.144} C_VEL
LIN {X 0,Y 134.737,Z 934.472,A -85,B 0,C 180,E1 -26301.415,E2 -26301.415} C_VEL
LIN {X 0,Y 139.332,Z 934.869,A -85,B 0,C 180,E1 -26303.798,E2 -26303.798} C_VEL
LIN {X 0,Y 149.372,Z 934.5,A -85,B 0,C 180,E1 -26308.067,E2 -26308.067} C_VEL
LIN {X 0,Y 160.167,Z 932.531,A -85,B 0,C 180,E1 -26311.772,E2 -26311.772} C_VEL
LIN {X 0,Y 167.27,Z 930.583,A -85,B 0,C 180,E1 -26313.818,E2 -26313.818} C_VEL
LIN {X 0,Y 167.691,Z 930.684,A -85,B 0,C 180,E1 -26314.502,E2 -26314.502} C_VEL
LIN {X 0,Y 154.939,Z 936.915,A -85,B 0,C 180,E1 -26317.452,E2 -26317.452} C_VEL
LIN {X 0,Y 146.675,Z 940.257,A -85,B 0,C 180,E1 -26319.94,E2 -26319.94} C_VEL
LIN {X 0,Y 136.481,Z 943.716,A -85,B 0,C 180,E1 -26323.863,E2 -26323.863} C_VEL
LIN {X 0,Y 127.605,Z 946.042,A -85,B 0,C 180,E1 -26328.624,E2 -26328.624} C_VEL
LIN {X 0,Y 120.083,Z 947.256,A -85,B 0,C 180,E1 -26334.173,E2 -26334.173} C_VEL
LIN {X 0,Y 114.321,Z 947.382,A -85,B 0,C 180,E1 -26340.535,E2 -26340.535} C_VEL
LIN {X 0,Y 110.021,Z 946.24,A -85,B 0,C 180,E1 -26349.67,E2 -26349.67} C_VEL
LIN {X 0,Y 108.026,Z 950.74,A -85,B 0,C 180,E1 -26354.91,E2 -26354.91} C_VEL
LIN {X 0,Y 107.308,Z 953.677,A -85,B 0,C 180,E1 -26359.235,E2 -26359.235} C_VEL
LIN {X 0,Y 107.273,Z 955.447,A -85,B 0,C 180,E1 -26362.465,E2 -26362.465} C_VEL
LIN {X 0,Y 107.53,Z 957.092,A -85,B 0,C 180,E1 -26366.247,E2 -26366.247} C_VEL
LIN {X 0,Y 108.04,Z 958.289,A -85,B 0,C 180,E1 -26369.994,E2 -26369.994} C_VEL
LIN {X 0,Y 107.392,Z 958.811,A -85,B 0,C 180,E1 -26373.747,E2 -26373.747} C_VEL
LIN {X 0,Y 106.816,Z 958.793,A -85,B 0,C 180,E1 -26379.276,E2 -26379.276} C_VEL
LIN {X 0,Y 107.137,Z 957.87,A -85,B 0,C 180,E1 -26385.206,E2 -26385.206} C_VEL
LIN {X 0,Y 109.309,Z 955.369,A -85,B 0,C 180,E1 -26392.685,E2 -26392.685} C_VEL
LIN {X 0,Y 110.25,Z 954.357,A -85,B 0,C 180,E1 -26394.663,E2 -26394.663} C_VEL
LIN {X 0,Y 111.262,Z 952.779,A -85,B 0,C 180,E1 -26397.564,E2 -26397.564} C_VEL
LIN {X 0,Y 111.932,Z 949.625,A -85,B 0,C 180,E1 -26402.39,E2 -26402.39} C_VEL
LIN {X 0,Y 113.36,Z 945.945,A -85,B 0,C 180,E1 -26407.013,E2 -26407.013} C_VEL
LIN {X 0,Y 115.48,Z 943.436,A -85,B 0,C 180,E1 -26409.477,E2 -26409.477} C_VEL
LIN {X 0,Y 122.929,Z 936.35,A -85,B 0,C 180,E1 -26414.448,E2 -26414.448} C_VEL
LIN {X 0,Y 129.884,Z 928.934,A -85,B 0,C 180,E1 -26418.067,E2 -26418.067} C_VEL
LIN {X 0,Y 137.471,Z 919.853,A -85,B 0,C 180,E1 -26421.22,E2 -26421.22} C_VEL
LIN {X 0,Y 144.098,Z 910.647,A -85,B 0,C 180,E1 -26423.578,E2 -26423.578} C_VEL
LIN {X 0,Y 150.329,Z 900.607,A -85,B 0,C 180,E1 -26425.478,E2 -26425.478} C_VEL
LIN {X 0,Y 156.046,Z 889.619,A -85,B 0,C 180,E1 -26427.009,E2 -26427.009} C_VEL
LIN {X 0,Y 161.124,Z 877.562,A -85,B 0,C 180,E1 -26428.238,E2 -26428.238} C_VEL
LIN {X 0,Y 165.153,Z 865.15,A -85,B 0,C 180,E1 -26429.156,E2 -26429.156} C_VEL
LIN {X 0,Y 168.059,Z 852.05,A -85,B 0,C 180,E1 -26429.88,E2 -26429.88} C_VEL
LIN {X 0,Y 169.195,Z 838.084,A -85,B 0,C 180,E1 -26431.032,E2 -26431.032} C_VEL
LIN {X 0,Y 169.605,Z 829.282,A -85,B 0,C 180,E1 -26431.815,E2 -26431.815} C_VEL
LIN {X 0,Y 168.016,Z 822.346,A -85,B 0,C 180,E1 -26434.529,E2 -26434.529} C_VEL
LIN {X 0,Y 166.562,Z 816.204,A -85,B 0,C 180,E1 -26437.582,E2 -26437.582} C_VEL
LIN {X 0,Y 165.155,Z 810.384,A -85,B 0,C 180,E1 -26441.798,E2 -26441.798} C_VEL
LIN {X 0,Y 164.459,Z 806.557,A -85,B 0,C 180,E1 -26446.489,E2 -26446.489} C_VEL
LIN {X 0,Y 164.44,Z 805.89,A -85,B 0,C 180,E1 -26447.661,E2 -26447.661} C_VEL
LIN {X 0,Y 164.663,Z 805.84,A -85,B 0,C 180,E1 -26451.48,E2 -26451.48} C_VEL
LIN {X 0,Y 165.564,Z 806.811,A -85,B 0,C 180,E1 -26455.257,E2 -26455.257} C_VEL
LIN {X 0,Y 167.318,Z 810.777,A -85,B 0,C 180,E1 -26459.67,E2 -26459.67} C_VEL
LIN {X 0,Y 169.132,Z 814.877,A -85,B 0,C 180,E1 -26462.766,E2 -26462.766} C_VEL
LIN {X 0,Y 171.262,Z 819.826,A -85,B 0,C 180,E1 -26465.705,E2 -26465.705} C_VEL
LIN {X 0,Y 171.801,Z 821.154,A -85,B 0,C 180,E1 -26466.363,E2 -26466.363} C_VEL
LIN {X 0,Y 170.143,Z 836.194,A -85,B 0,C 180,E1 -26467.254,E2 -26467.254} C_VEL
LIN {X 0,Y 167.647,Z 848.377,A -85,B 0,C 180,E1 -26468.266,E2 -26468.266} C_VEL
LIN {X 0,Y 163.944,Z 860.795,A -85,B 0,C 180,E1 -26469.632,E2 -26469.632} C_VEL
LIN {X 0,Y 159.283,Z 872.509,A -85,B 0,C 180,E1 -26471.315,E2 -26471.315} C_VEL
LIN {X 0,Y 153.495,Z 883.887,A -85,B 0,C 180,E1 -26473.512,E2 -26473.512} C_VEL
LIN {X 0,Y 147.886,Z 892.976,A -85,B 0,C 180,E1 -26475.79,E2 -26475.79} C_VEL
LIN {X 0,Y 142.262,Z 900.745,A -85,B 0,C 180,E1 -26478.297,E2 -26478.297} C_VEL
LIN {X 0,Y 135.938,Z 908.278,A -85,B 0,C 180,E1 -26481.484,E2 -26481.484} C_VEL
LIN {X 0,Y 129.266,Z 914.974,A -85,B 0,C 180,E1 -26485.301,E2 -26485.301} C_VEL
LIN {X 0,Y 122.159,Z 921.085,A -85,B 0,C 180,E1 -26490.359,E2 -26490.359} C_VEL
LIN {X 0,Y 116.397,Z 925.191,A -85,B 0,C 180,E1 -26495.41,E2 -26495.41} C_VEL
LIN {X 0,Y 111.49,Z 927.994,A -85,B 0,C 180,E1 -26500.857,E2 -26500.857} C_VEL
LIN {X 0,Y 108.257,Z 929.42,A -85,B 0,C 180,E1 -26505.572,E2 -26505.572} C_VEL
LIN {X 0,Y 106.517,Z 929.955,A -85,B 0,C 180,E1 -26508.723,E2 -26508.723} C_VEL
LIN {X 0,Y 104.286,Z 930.173,A -85,B 0,C 180,E1 -26513.971,E2 -26513.971} C_VEL
LIN {X 0,Y 102.506,Z 929.296,A -85,B 0,C 180,E1 -26521.326,E2 -26521.326} C_VEL
LIN {X 0,Y 102.131,Z 928.128,A -85,B 0,C 180,E1 -26525.621,E2 -26525.621} C_VEL
LIN {X 0,Y 102.716,Z 924.886,A -85,B 0,C 180,E1 -26533.319,E2 -26533.319} C_VEL
LIN {X 0,Y 104.588,Z 920.335,A -85,B 0,C 180,E1 -26540.335,E2 -26540.335} C_VEL
LIN {X 0,Y 107.762,Z 914.04,A -85,B 0,C 180,E1 -26547.202,E2 -26547.202} C_VEL
LIN {X 0,Y 111.318,Z 907.126,A -85,B 0,C 180,E1 -26552.719,E2 -26552.719} C_VEL
LIN {X 0,Y 115.626,Z 898.516,A -85,B 0,C 180,E1 -26557.866,E2 -26557.866} C_VEL
LIN {X 0,Y 119.706,Z 889.745,A -85,B 0,C 180,E1 -26561.863,E2 -26561.863} C_VEL
LIN {X 0,Y 123.966,Z 879.4,A -85,B 0,C 180,E1 -26565.464,E2 -26565.464} C_VEL
LIN {X 0,Y 127.872,Z 868.277,A -85,B 0,C 180,E1 -26568.428,E2 -26568.428} C_VEL
LIN {X 0,Y 131.365,Z 856.555,A -85,B 0,C 180,E1 -26570.764,E2 -26570.764} C_VEL
LIN {X 0,Y 133.919,Z 845.165,A -85,B 0,C 180,E1 -26572.487,E2 -26572.487} C_VEL
LIN {X 0,Y 136.065,Z 831.24,A -85,B 0,C 180,E1 -26574.012,E2 -26574.012} C_VEL
LIN {X 0,Y 137.206,Z 817.923,A -85,B 0,C 180,E1 -26574.942,E2 -26574.942} C_VEL
LIN {X 0,Y 138.295,Z 797.887,A -85,B 0,C 180,E1 -26576.037,E2 -26576.037} C_VEL
LIN {X 0,Y 132.003,Z 785.002,A -85,B 0,C 180,E1 -26579.819,E2 -26579.819} C_VEL
LIN {X 0,Y 126.196,Z 774.644,A -85,B 0,C 180,E1 -26583.761,E2 -26583.761} C_VEL
LIN {X 0,Y 121.45,Z 767.173,A -85,B 0,C 180,E1 -26587.409,E2 -26587.409} C_VEL
LIN {X 0,Y 119.367,Z 769.707,A -85,B 0,C 180,E1 -26588.55,E2 -26588.55} C_VEL
LIN {X 0,Y 117.623,Z 771.05,A -85,B 0,C 180,E1 -26589.641,E2 -26589.641} C_VEL
LIN {X 0,Y 115.91,Z 775.02,A -85,B 0,C 180,E1 -26590.446,E2 -26590.446} C_VEL
LIN {X 0,Y 114.58,Z 777.641,A -85,B 0,C 180,E1 -26591.157,E2 -26591.157} C_VEL
LIN {X 0,Y 112.938,Z 780.662,A -85,B 0,C 180,E1 -26592.142,E2 -26592.142} C_VEL
LIN {X 0,Y 112.148,Z 781.804,A -85,B 0,C 180,E1 -26592.86,E2 -26592.86} C_VEL
LIN {X 0,Y 111.526,Z 785,A -85,B 0,C 180,E1 -26593.739,E2 -26593.739} C_VEL
LIN {X 0,Y 110.839,Z 793.172,A -85,B 0,C 180,E1 -26594.934,E2 -26594.934} C_VEL
LIN {X 0,Y 108.989,Z 822.299,A -85,B 0,C 180,E1 -26598.163,E2 -26598.163} C_VEL
LIN {X 0,Y 107.74,Z 835.583,A -85,B 0,C 180,E1 -26600.196,E2 -26600.196} C_VEL
LIN {X 0,Y 106.429,Z 846.614,A -85,B 0,C 180,E1 -26602.42,E2 -26602.42} C_VEL
LIN {X 0,Y 105.236,Z 856.176,A -85,B 0,C 180,E1 -26604.829,E2 -26604.829} C_VEL
LIN {X 0,Y 104.193,Z 864.481,A -85,B 0,C 180,E1 -26607.342,E2 -26607.342} C_VEL
LIN {X 0,Y 102.86,Z 874.2,A -85,B 0,C 180,E1 -26610.867,E2 -26610.867} C_VEL
LIN {X 0,Y 101.865,Z 883.204,A -85,B 0,C 180,E1 -26614.769,E2 -26614.769} C_VEL
LIN {X 0,Y 101.209,Z 890.818,A -85,B 0,C 180,E1 -26618.619,E2 -26618.619} C_VEL
LIN {X 0,Y 100.878,Z 899.47,A -85,B 0,C 180,E1 -26623.818,E2 -26623.818} C_VEL
LIN {X 0,Y 101.179,Z 906.752,A -85,B 0,C 180,E1 -26628.987,E2 -26628.987} C_VEL
LIN {X 0,Y 102.256,Z 913.022,A -85,B 0,C 180,E1 -26634.082,E2 -26634.082} C_VEL
LIN {X 0,Y 104.564,Z 919.302,A -85,B 0,C 180,E1 -26639.999,E2 -26639.999} C_VEL
LIN {X 0,Y 107.877,Z 924.457,A -85,B 0,C 180,E1 -26645.607,E2 -26645.607} C_VEL
LIN {X 0,Y 112.163,Z 928.629,A -85,B 0,C 180,E1 -26650.834,E2 -26650.834} C_VEL
LIN {X 0,Y 116.219,Z 931.29,A -85,B 0,C 180,E1 -26654.618,E2 -26654.618} C_VEL
LIN {X 0,Y 123.504,Z 934.265,A -85,B 0,C 180,E1 -26659.964,E2 -26659.964} C_VEL
LIN {X 0,Y 132.736,Z 936.062,A -85,B 0,C 180,E1 -26665.06,E2 -26665.06} C_VEL
LIN {X 0,Y 137.784,Z 936.407,A -85,B 0,C 180,E1 -26667.326,E2 -26667.326} C_VEL
LIN {X 0,Y 148.524,Z 935.905,A -85,B 0,C 180,E1 -26671.366,E2 -26671.366} C_VEL
LIN {X 0,Y 155.395,Z 934.914,A -85,B 0,C 180,E1 -26673.502,E2 -26673.502} C_VEL
LIN {X 0,Y 153.66,Z 935.867,A -85,B 0,C 180,E1 -26674.58,E2 -26674.58} C_VEL
LIN {X 0,Y 142.238,Z 939.976,A -85,B 0,C 180,E1 -26677.756,E2 -26677.756} C_VEL
LIN {X 0,Y 131.675,Z 943.002,A -85,B 0,C 180,E1 -26681.643,E2 -26681.643} C_VEL
LIN {X 0,Y 122.417,Z 944.909,A -85,B 0,C 180,E1 -26686.449,E2 -26686.449} C_VEL
LIN {X 0,Y 114.496,Z 945.669,A -85,B 0,C 180,E1 -26692.127,E2 -26692.127} C_VEL
LIN {X 0,Y 111.164,Z 945.752,A -85,B 0,C 180,E1 -26695.313,E2 -26695.313} C_VEL
LIN {X 0,Y 106.089,Z 945.034,A -85,B 0,C 180,E1 -26702.366,E2 -26702.366} C_VEL
LIN {X 0,Y 103.86,Z 944.117,A -85,B 0,C 180,E1 -26707.621,E2 -26707.621} C_VEL
LIN {X 0,Y 101.201,Z 949.346,A -85,B 0,C 180,E1 -26713.866,E2 -26713.866} C_VEL
LIN {X 0,Y 100.341,Z 952.489,A -85,B 0,C 180,E1 -26718.687,E2 -26718.687} C_VEL
LIN {X 0,Y 100.463,Z 955.88,A -85,B 0,C 180,E1 -26725.983,E2 -26725.983} C_VEL
LIN {X 0,Y 100.976,Z 957.124,A -85,B 0,C 180,E1 -26729.994,E2 -26729.994} C_VEL
LIN {X 0,Y 100.307,Z 957.7,A -85,B 0,C 180,E1 -26734.012,E2 -26734.012} C_VEL
LIN {X 0,Y 99.79,Z 957.757,A -85,B 0,C 180,E1 -26739.603,E2 -26739.603} C_VEL
LIN {X 0,Y 100.232,Z 956.901,A -85,B 0,C 180,E1 -26746.282,E2 -26746.282} C_VEL
LIN {X 0,Y 102.718,Z 954.522,A -85,B 0,C 180,E1 -26754.231,E2 -26754.231} C_VEL
LIN {X 0,Y 106.007,Z 951.709,A -85,B 0,C 180,E1 -26759.81,E2 -26759.81} C_VEL
LIN {X 0,Y 110.479,Z 947.989,A -85,B 0,C 180,E1 -26764.919,E2 -26764.919} C_VEL
LIN {X 0,Y 115.48,Z 943.436,A -85,B 0,C 180,E1 -26769.477,E2 -26769.477} C_VEL
LIN {X 0,Y 117.8,Z 940.777,A -85,B 0,C 180,E1 -26771.814,E2 -26771.814} C_VEL
LIN {X 0,Y 120.567,Z 936.036,A -85,B 0,C 180,E1 -26775.793,E2 -26775.793} C_VEL
LIN {X 0,Y 123.782,Z 930.731,A -85,B 0,C 180,E1 -26779.402,E2 -26779.402} C_VEL
LIN {X 0,Y 126.676,Z 927.194,A -85,B 0,C 180,E1 -26781.1,E2 -26781.1} C_VEL
LIN {X 0,Y 134.51,Z 918.212,A -85,B 0,C 180,E1 -26784.074,E2 -26784.074} C_VEL
LIN {X 0,Y 140.012,Z 910.904,A -85,B 0,C 180,E1 -26785.909,E2 -26785.909} C_VEL
LIN {X 0,Y 147.171,Z 899.988,A -85,B 0,C 180,E1 -26787.947,E2 -26787.947} C_VEL
LIN {X 0,Y 153.068,Z 889.141,A -85,B 0,C 180,E1 -26789.409,E2 -26789.409} C_VEL
LIN {X 0,Y 158.319,Z 877.144,A -85,B 0,C 180,E1 -26790.587,E2 -26790.587} C_VEL
LIN {X 0,Y 162.651,Z 864.251,A -85,B 0,C 180,E1 -26791.507,E2 -26791.507} C_VEL
LIN {X 0,Y 165.516,Z 851.908,A -85,B 0,C 180,E1 -26792.194,E2 -26792.194} C_VEL
LIN {X 0,Y 166.824,Z 838.112,A -85,B 0,C 180,E1 -26793.374,E2 -26793.374} C_VEL
LIN {X 0,Y 167.137,Z 832.975,A -85,B 0,C 180,E1 -26793.83,E2 -26793.83} C_VEL
LIN {X 0,Y 165.979,Z 827.086,A -85,B 0,C 180,E1 -26796.281,E2 -26796.281} C_VEL
LIN {X 0,Y 164.837,Z 821.612,A -85,B 0,C 180,E1 -26799.224,E2 -26799.224} C_VEL
LIN {X 0,Y 163.971,Z 817.053,A -85,B 0,C 180,E1 -26802.541,E2 -26802.541} C_VEL
LIN {X 0,Y 163.482,Z 813.295,A -85,B 0,C 180,E1 -26807.195,E2 -26807.195} C_VEL
LIN {X 0,Y 163.475,Z 812.841,A -85,B 0,C 180,E1 -26808.408,E2 -26808.408} C_VEL
LIN {X 0,Y 163.71,Z 812.877,A -85,B 0,C 180,E1 -26811.43,E2 -26811.43} C_VEL
LIN {X 0,Y 164.415,Z 813.655,A -85,B 0,C 180,E1 -26814.681,E2 -26814.681} C_VEL
LIN {X 0,Y 165.986,Z 817.478,A -85,B 0,C 180,E1 -26819,E2 -26819} C_VEL
LIN {X 0,Y 168.072,Z 822.58,A -85,B 0,C 180,E1 -26822.783,E2 -26822.783} C_VEL
LIN {X 0,Y 169.072,Z 825.56,A -85,B 0,C 180,E1 -26824.354,E2 -26824.354} C_VEL
LIN {X 0,Y 167.322,Z 838.681,A -85,B 0,C 180,E1 -26825.154,E2 -26825.154} C_VEL
LIN {X 0,Y 164.197,Z 852.2,A -85,B 0,C 180,E1 -26826.29,E2 -26826.29} C_VEL
LIN {X 0,Y 160.227,Z 864.232,A -85,B 0,C 180,E1 -26827.665,E2 -26827.665} C_VEL
LIN {X 0,Y 154.994,Z 876.147,A -85,B 0,C 180,E1 -26829.46,E2 -26829.46} C_VEL
LIN {X 0,Y 148.881,Z 887.189,A -85,B 0,C 180,E1 -26831.64,E2 -26831.64} C_VEL
LIN {X 0,Y 142.135,Z 897.102,A -85,B 0,C 180,E1 -26834.314,E2 -26834.314} C_VEL
LIN {X 0,Y 134.585,Z 906.308,A -85,B 0,C 180,E1 -26837.651,E2 -26837.651} C_VEL
LIN {X 0,Y 126.754,Z 914.19,A -85,B 0,C 180,E1 -26841.702,E2 -26841.702} C_VEL
LIN {X 0,Y 120.634,Z 919.443,A -85,B 0,C 180,E1 -26845.456,E2 -26845.456} C_VEL
LIN {X 0,Y 114.046,Z 924.281,A -85,B 0,C 180,E1 -26850.386,E2 -26850.386} C_VEL
LIN {X 0,Y 108.331,Z 927.714,A -85,B 0,C 180,E1 -26855.725,E2 -26855.725} C_VEL
LIN {X 0,Y 102.188,Z 930.411,A -85,B 0,C 180,E1 -26863.454,E2 -26863.454} C_VEL
LIN {X 0,Y 98.615,Z 931.223,A -85,B 0,C 180,E1 -26870.112,E2 -26870.112} C_VEL
LIN {X 0,Y 96.947,Z 931.116,A -85,B 0,C 180,E1 -26874.561,E2 -26874.561} C_VEL
LIN {X 0,Y 95.342,Z 929.926,A -85,B 0,C 180,E1 -26882.2,E2 -26882.2} C_VEL
LIN {X 0,Y 95.116,Z 928.059,A -85,B 0,C 180,E1 -26888.326,E2 -26888.326} C_VEL
LIN {X 0,Y 95.992,Z 924.925,A -85,B 0,C 180,E1 -26895.174,E2 -26895.174} C_VEL
LIN {X 0,Y 97.911,Z 920.687,A -85,B 0,C 180,E1 -26901.752,E2 -26901.752} C_VEL
LIN {X 0,Y 100.855,Z 915.205,A -85,B 0,C 180,E1 -26908.009,E2 -26908.009} C_VEL
LIN {X 0,Y 104.595,Z 908.34,A -85,B 0,C 180,E1 -26913.858,E2 -26913.858} C_VEL
LIN {X 0,Y 109.113,Z 899.773,A -85,B 0,C 180,E1 -26919.272,E2 -26919.272} C_VEL
LIN {X 0,Y 113.438,Z 891.033,A -85,B 0,C 180,E1 -26923.44,E2 -26923.44} C_VEL
LIN {X 0,Y 117.471,Z 881.903,A -85,B 0,C 180,E1 -26926.813,E2 -26926.813} C_VEL
LIN {X 0,Y 121.538,Z 871.175,A -85,B 0,C 180,E1 -26929.865,E2 -26929.865} C_VEL
LIN {X 0,Y 125.143,Z 859.939,A -85,B 0,C 180,E1 -26932.282,E2 -26932.282} C_VEL
LIN {X 0,Y 128.225,Z 847.663,A -85,B 0,C 180,E1 -26934.277,E2 -26934.277} C_VEL
LIN {X 0,Y 130.557,Z 834.242,A -85,B 0,C 180,E1 -26935.831,E2 -26935.831} C_VEL
LIN {X 0,Y 131.82,Z 821.63,A -85,B 0,C 180,E1 -26936.826,E2 -26936.826} C_VEL
LIN {X 0,Y 133.09,Z 800.453,A -85,B 0,C 180,E1 -26938.021,E2 -26938.021} C_VEL
LIN {X 0,Y 127.565,Z 788.741,A -85,B 0,C 180,E1 -26941.711,E2 -26941.711} C_VEL
LIN {X 0,Y 121.318,Z 777.551,A -85,B 0,C 180,E1 -26946.381,E2 -26946.381} C_VEL
LIN {X 0,Y 120.246,Z 776.206,A -85,B 0,C 180,E1 -26947.224,E2 -26947.224} C_VEL
LIN {X 0,Y 115.749,Z 784.571,A -85,B 0,C 180,E1 -26949.422,E2 -26949.422} C_VEL
LIN {X 0,Y 113.912,Z 787.132,A -85,B 0,C 180,E1 -26950.501,E2 -26950.501} C_VEL
LIN {X 0,Y 111.084,Z 796.498,A -85,B 0,C 180,E1 -26951.571,E2 -26951.571} C_VEL
LIN {X 0,Y 107.092,Z 809.701,A -85,B 0,C 180,E1 -26953.234,E2 -26953.234} C_VEL
LIN {X 0,Y 104.504,Z 816.186,A -85,B 0,C 180,E1 -26954.737,E2 -26954.737} C_VEL
LIN {X 0,Y 103.007,Z 818.753,A -85,B 0,C 180,E1 -26955.966,E2 -26955.966} C_VEL
LIN {X 0,Y 102.276,Z 821.179,A -85,B 0,C 180,E1 -26956.965,E2 -26956.965} C_VEL
LIN {X 0,Y 101.466,Z 827.527,A -85,B 0,C 180,E1 -26958.388,E2 -26958.388} C_VEL
LIN {X 0,Y 99.68,Z 843.86,A -85,B 0,C 180,E1 -26961.585,E2 -26961.585} C_VEL
LIN {X 0,Y 98.042,Z 856.736,A -85,B 0,C 180,E1 -26965.007,E2 -26965.007} C_VEL
LIN {X 0,Y 96.735,Z 866.512,A -85,B 0,C 180,E1 -26968.214,E2 -26968.214} C_VEL
LIN {X 0,Y 95.496,Z 876.146,A -85,B 0,C 180,E1 -26972.035,E2 -26972.035} C_VEL
LIN {X 0,Y 94.638,Z 884.303,A -85,B 0,C 180,E1 -26975.892,E2 -26975.892} C_VEL
LIN {X 0,Y 94.065,Z 892.34,A -85,B 0,C 180,E1 -26980.353,E2 -26980.353} C_VEL
LIN {X 0,Y 93.904,Z 900.995,A -85,B 0,C 180,E1 -26986.033,E2 -26986.033} C_VEL
LIN {X 0,Y 94.53,Z 908.112,A -85,B 0,C 180,E1 -26991.448,E2 -26991.448} C_VEL
LIN {X 0,Y 96.4,Z 915.392,A -85,B 0,C 180,E1 -26997.91,E2 -26997.91} C_VEL
LIN {X 0,Y 98.496,Z 920.08,A -85,B 0,C 180,E1 -27002.513,E2 -27002.513} C_VEL
LIN {X 0,Y 101.913,Z 924.994,A -85,B 0,C 180,E1 -27007.927,E2 -27007.927} C_VEL
LIN {X 0,Y 106.643,Z 929.334,A -85,B 0,C 180,E1 -27013.335,E2 -27013.335} C_VEL
LIN {X 0,Y 112.361,Z 932.759,A -85,B 0,C 180,E1 -27018.224,E2 -27018.224} C_VEL
LIN {X 0,Y 121.23,Z 935.94,A -85,B 0,C 180,E1 -27023.941,E2 -27023.941} C_VEL
LIN {X 0,Y 131.359,Z 937.654,A -85,B 0,C 180,E1 -27028.784,E2 -27028.784} C_VEL
LIN {X 0,Y 136.812,Z 937.94,A -85,B 0,C 180,E1 -27030.91,E2 -27030.91} C_VEL
LIN {X 0,Y 142.422,Z 937.77,A -85,B 0,C 180,E1 -27032.875,E2 -27032.875} C_VEL
LIN {X 0,Y 143.764,Z 937.94,A -85,B 0,C 180,E1 -27033.786,E2 -27033.786} C_VEL
LIN {X 0,Y 132.422,Z 941.026,A -85,B 0,C 180,E1 -27037.235,E2 -27037.235} C_VEL
LIN {X 0,Y 122.115,Z 943.028,A -85,B 0,C 180,E1 -27041.56,E2 -27041.56} C_VEL
LIN {X 0,Y 113.041,Z 943.956,A -85,B 0,C 180,E1 -27046.845,E2 -27046.845} C_VEL
LIN {X 0,Y 105.551,Z 943.912,A -85,B 0,C 180,E1 -27053.177,E2 -27053.177} C_VEL
LIN {X 0,Y 100.063,Z 942.882,A -85,B 0,C 180,E1 -27060.544,E2 -27060.544} C_VEL
LIN {X 0,Y 97.804,Z 942.01,A -85,B 0,C 180,E1 -27065.447,E2 -27065.447} C_VEL
LIN {X 0,Y 94.407,Z 947.936,A -85,B 0,C 180,E1 -27072.669,E2 -27072.669} C_VEL
LIN {X 0,Y 93.343,Z 951.337,A -85,B 0,C 180,E1 -27078.177,E2 -27078.177} C_VEL
LIN {X 0,Y 93.398,Z 954.661,A -85,B 0,C 180,E1 -27085.678,E2 -27085.678} C_VEL
LIN {X 0,Y 93.91,Z 955.951,A -85,B 0,C 180,E1 -27089.994,E2 -27089.994} C_VEL
LIN {X 0,Y 93.224,Z 956.563,A -85,B 0,C 180,E1 -27094.317,E2 -27094.317} C_VEL
LIN {X 0,Y 92.762,Z 956.721,A -85,B 0,C 180,E1 -27099.961,E2 -27099.961} C_VEL
LIN {X 0,Y 93.38,Z 955.935,A -85,B 0,C 180,E1 -27107.514,E2 -27107.514} C_VEL
LIN {X 0,Y 96.223,Z 953.647,A -85,B 0,C 180,E1 -27115.984,E2 -27115.984} C_VEL
LIN {X 0,Y 100.492,Z 950.475,A -85,B 0,C 180,E1 -27122.692,E2 -27122.692} C_VEL
LIN {X 0,Y 106.455,Z 945.937,A -85,B 0,C 180,E1 -27128.834,E2 -27128.834} C_VEL
LIN {X 0,Y 112.369,Z 940.977,A -85,B 0,C 180,E1 -27133.463,E2 -27133.463} C_VEL
LIN {X 0,Y 120.299,Z 933.689,A -85,B 0,C 180,E1 -27138.14,E2 -27138.14} C_VEL
LIN {X 0,Y 126.676,Z 927.194,A -85,B 0,C 180,E1 -27141.1,E2 -27141.1} C_VEL
LIN {X 0,Y 129.621,Z 923.516,A -85,B 0,C 180,E1 -27142.699,E2 -27142.699} C_VEL
LIN {X 0,Y 133.292,Z 917.265,A -85,B 0,C 180,E1 -27145.669,E2 -27145.669} C_VEL
LIN {X 0,Y 137.001,Z 910.543,A -85,B 0,C 180,E1 -27148.31,E2 -27148.31} C_VEL
LIN {X 0,Y 139.867,Z 906.109,A -85,B 0,C 180,E1 -27149.382,E2 -27149.382} C_VEL
LIN {X 0,Y 147.295,Z 894.288,A -85,B 0,C 180,E1 -27151.242,E2 -27151.242} C_VEL
LIN {X 0,Y 153.444,Z 882.268,A -85,B 0,C 180,E1 -27152.54,E2 -27152.54} C_VEL
LIN {X 0,Y 158.354,Z 869.954,A -85,B 0,C 180,E1 -27153.521,E2 -27153.521} C_VEL
LIN {X 0,Y 162.306,Z 856.551,A -85,B 0,C 180,E1 -27154.285,E2 -27154.285} C_VEL
LIN {X 0,Y 163.581,Z 849.824,A -85,B 0,C 180,E1 -27154.756,E2 -27154.756} C_VEL
LIN {X 0,Y 164.917,Z 836.65,A -85,B 0,C 180,E1 -27155.934,E2 -27155.934} C_VEL
LIN {X 0,Y 163.868,Z 830.481,A -85,B 0,C 180,E1 -27158.785,E2 -27158.785} C_VEL
LIN {X 0,Y 163.326,Z 827.232,A -85,B 0,C 180,E1 -27160.741,E2 -27160.741} C_VEL
LIN {X 0,Y 162.762,Z 823.458,A -85,B 0,C 180,E1 -27163.577,E2 -27163.577} C_VEL
LIN {X 0,Y 162.526,Z 820.055,A -85,B 0,C 180,E1 -27167.927,E2 -27167.927} C_VEL
LIN {X 0,Y 162.607,Z 819.76,A -85,B 0,C 180,E1 -27170.045,E2 -27170.045} C_VEL
LIN {X 0,Y 163.328,Z 820.607,A -85,B 0,C 180,E1 -27174.227,E2 -27174.227} C_VEL
LIN {X 0,Y 164.673,Z 824.199,A -85,B 0,C 180,E1 -27178.32,E2 -27178.32} C_VEL
LIN {X 0,Y 166.377,Z 828.882,A -85,B 0,C 180,E1 -27181.816,E2 -27181.816} C_VEL
LIN {X 0,Y 166.573,Z 829.514,A -85,B 0,C 180,E1 -27182.192,E2 -27182.192} C_VEL
LIN {X 0,Y 164.384,Z 843.191,A -85,B 0,C 180,E1 -27183.108,E2 -27183.108} C_VEL
LIN {X 0,Y 161.069,Z 855.714,A -85,B 0,C 180,E1 -27184.219,E2 -27184.219} C_VEL
LIN {X 0,Y 156.955,Z 866.971,A -85,B 0,C 180,E1 -27185.522,E2 -27185.522} C_VEL
LIN {X 0,Y 151.44,Z 878.689,A -85,B 0,C 180,E1 -27187.303,E2 -27187.303} C_VEL
LIN {X 0,Y 145.137,Z 889.269,A -85,B 0,C 180,E1 -27189.41,E2 -27189.41} C_VEL
LIN {X 0,Y 138.206,Z 898.898,A -85,B 0,C 180,E1 -27192.007,E2 -27192.007} C_VEL
LIN {X 0,Y 130.969,Z 907.274,A -85,B 0,C 180,E1 -27195.023,E2 -27195.023} C_VEL
LIN {X 0,Y 124.021,Z 914.041,A -85,B 0,C 180,E1 -27198.36,E2 -27198.36} C_VEL
LIN {X 0,Y 117.325,Z 919.579,A -85,B 0,C 180,E1 -27202.05,E2 -27202.05} C_VEL
LIN {X 0,Y 110.268,Z 924.535,A -85,B 0,C 180,E1 -27206.849,E2 -27206.849} C_VEL
LIN {X 0,Y 105.896,Z 927.16,A -85,B 0,C 180,E1 -27210.383,E2 -27210.383} C_VEL
LIN {X 0,Y 101.936,Z 929.174,A -85,B 0,C 180,E1 -27214.185,E2 -27214.185} C_VEL
LIN {X 0,Y 96.277,Z 931.408,A -85,B 0,C 180,E1 -27221.071,E2 -27221.071} C_VEL
LIN {X 0,Y 92.784,Z 932.185,A -85,B 0,C 180,E1 -27227.032,E2 -27227.032} C_VEL
LIN {X 0,Y 90.752,Z 932.247,A -85,B 0,C 180,E1 -27231.727,E2 -27231.727} C_VEL
LIN {X 0,Y 89.276,Z 931.804,A -85,B 0,C 180,E1 -27236.569,E2 -27236.569} C_VEL
LIN {X 0,Y 88.373,Z 930.913,A -85,B 0,C 180,E1 -27241.508,E2 -27241.508} C_VEL
LIN {X 0,Y 88.045,Z 929.584,A -85,B 0,C 180,E1 -27246.485,E2 -27246.485} C_VEL
LIN {X 0,Y 88.432,Z 927.288,A -85,B 0,C 180,E1 -27252.496,E2 -27252.496} C_VEL
LIN {X 0,Y 89.731,Z 924.083,A -85,B 0,C 180,E1 -27258.715,E2 -27258.715} C_VEL
LIN {X 0,Y 92.257,Z 919.269,A -85,B 0,C 180,E1 -27265.638,E2 -27265.638} C_VEL
LIN {X 0,Y 95.809,Z 913.162,A -85,B 0,C 180,E1 -27272.108,E2 -27272.108} C_VEL
LIN {X 0,Y 100.206,Z 905.515,A -85,B 0,C 180,E1 -27278.07,E2 -27278.07} C_VEL
LIN {X 0,Y 104.479,Z 897.732,A -85,B 0,C 180,E1 -27282.634,E2 -27282.634} C_VEL
LIN {X 0,Y 109.335,Z 887.947,A -85,B 0,C 180,E1 -27287.012,E2 -27287.012} C_VEL
LIN {X 0,Y 113.735,Z 878.005,A -85,B 0,C 180,E1 -27290.345,E2 -27290.345} C_VEL
LIN {X 0,Y 117.943,Z 866.566,A -85,B 0,C 180,E1 -27293.257,E2 -27293.257} C_VEL
LIN {X 0,Y 121.76,Z 853.812,A -85,B 0,C 180,E1 -27295.657,E2 -27295.657} C_VEL
LIN {X 0,Y 124.565,Z 840.799,A -85,B 0,C 180,E1 -27297.421,E2 -27297.421} C_VEL
LIN {X 0,Y 126.371,Z 827.844,A -85,B 0,C 180,E1 -27298.655,E2 -27298.655} C_VEL
LIN {X 0,Y 128.06,Z 803.005,A -85,B 0,C 180,E1 -27300.166,E2 -27300.166} C_VEL
LIN {X 0,Y 123.109,Z 792.374,A -85,B 0,C 180,E1 -27303.783,E2 -27303.783} C_VEL
LIN {X 0,Y 120.134,Z 786.798,A -85,B 0,C 180,E1 -27306.155,E2 -27306.155} C_VEL
LIN {X 0,Y 119.814,Z 786.682,A -85,B 0,C 180,E1 -27306.374,E2 -27306.374} C_VEL
LIN {X 0,Y 116.643,Z 791.647,A -85,B 0,C 180,E1 -27307.964,E2 -27307.964} C_VEL
LIN {X 0,Y 110.991,Z 810.212,A -85,B 0,C 180,E1 -27309.895,E2 -27309.895} C_VEL
LIN {X 0,Y 107.942,Z 818.188,A -85,B 0,C 180,E1 -27311.323,E2 -27311.323} C_VEL
LIN {X 0,Y 105.746,Z 822.417,A -85,B 0,C 180,E1 -27312.655,E2 -27312.655} C_VEL
LIN {X 0,Y 104.089,Z 825.09,A -85,B 0,C 180,E1 -27313.811,E2 -27313.811} C_VEL
LIN {X 0,Y 99.382,Z 837.654,A -85,B 0,C 180,E1 -27316.058,E2 -27316.058} C_VEL
LIN {X 0,Y 95.849,Z 844.45,A -85,B 0,C 180,E1 -27318.033,E2 -27318.033} C_VEL
LIN {X 0,Y 94.03,Z 846.853,A -85,B 0,C 180,E1 -27319.412,E2 -27319.412} C_VEL
LIN {X 0,Y 93.135,Z 847.82,A -85,B 0,C 180,E1 -27320.272,E2 -27320.272} C_VEL
LIN {X 0,Y 92.071,Z 849.129,A -85,B 0,C 180,E1 -27322.037,E2 -27322.037} C_VEL
LIN {X 0,Y 91.524,Z 852.108,A -85,B 0,C 180,E1 -27323.478,E2 -27323.478} C_VEL
LIN {X 0,Y 89.706,Z 865.628,A -85,B 0,C 180,E1 -27328.096,E2 -27328.096} C_VEL
LIN {X 0,Y 88.305,Z 876.521,A -85,B 0,C 180,E1 -27332.765,E2 -27332.765} C_VEL
LIN {X 0,Y 87.446,Z 885.826,A -85,B 0,C 180,E1 -27337.557,E2 -27337.557} C_VEL
LIN {X 0,Y 87,Z 893.781,A -85,B 0,C 180,E1 -27342.365,E2 -27342.365} C_VEL
LIN {X 0,Y 87.104,Z 902.391,A -85,B 0,C 180,E1 -27348.562,E2 -27348.562} C_VEL
LIN {X 0,Y 88.106,Z 909.322,A -85,B 0,C 180,E1 -27354.277,E2 -27354.277} C_VEL
LIN {X 0,Y 89.991,Z 915.542,A -85,B 0,C 180,E1 -27359.999,E2 -27359.999} C_VEL
LIN {X 0,Y 93.335,Z 921.754,A -85,B 0,C 180,E1 -27366.485,E2 -27366.485} C_VEL
LIN {X 0,Y 97.777,Z 926.942,A -85,B 0,C 180,E1 -27372.452,E2 -27372.452} C_VEL
LIN {X 0,Y 103.377,Z 931.187,A -85,B 0,C 180,E1 -27377.847,E2 -27377.847} C_VEL
LIN {X 0,Y 109.786,Z 934.519,A -85,B 0,C 180,E1 -27382.587,E2 -27382.587} C_VEL
LIN {X 0,Y 119.604,Z 937.603,A -85,B 0,C 180,E1 -27388.039,E2 -27388.039} C_VEL
LIN {X 0,Y 130.593,Z 939.239,A -85,B 0,C 180,E1 -27392.558,E2 -27392.558} C_VEL
LIN {X 0,Y 131.722,Z 939.296,A -85,B 0,C 180,E1 -27392.952,E2 -27392.952} C_VEL
LIN {X 0,Y 130.16,Z 939.911,A -85,B 0,C 180,E1 -27394.124,E2 -27394.124} C_VEL
LIN {X 0,Y 122.756,Z 941.143,A -85,B 0,C 180,E1 -27396.716,E2 -27396.716} C_VEL
LIN {X 0,Y 112.672,Z 942.224,A -85,B 0,C 180,E1 -27401.531,E2 -27401.531} C_VEL
LIN {X 0,Y 103.861,Z 942.31,A -85,B 0,C 180,E1 -27407.408,E2 -27407.408} C_VEL
LIN {X 0,Y 96.866,Z 941.433,A -85,B 0,C 180,E1 -27414.512,E2 -27414.512} C_VEL
LIN {X 0,Y 92.011,Z 939.744,A -85,B 0,C 180,E1 -27422.87,E2 -27422.87} C_VEL
LIN {X 0,Y 87.672,Z 946.507,A -85,B 0,C 180,E1 -27431.291,E2 -27431.291} C_VEL
LIN {X 0,Y 86.357,Z 950.155,A -85,B 0,C 180,E1 -27437.578,E2 -27437.578} C_VEL
LIN {X 0,Y 86.337,Z 953.43,A -85,B 0,C 180,E1 -27445.324,E2 -27445.324} C_VEL
LIN {X 0,Y 86.842,Z 954.772,A -85,B 0,C 180,E1 -27449.993,E2 -27449.993} C_VEL
LIN {X 0,Y 86.141,Z 955.422,A -85,B 0,C 180,E1 -27454.673,E2 -27454.673} C_VEL
LIN {X 0,Y 85.735,Z 955.675,A -85,B 0,C 180,E1 -27460.368,E2 -27460.368} C_VEL
LIN {X 0,Y 86.588,Z 954.973,A -85,B 0,C 180,E1 -27468.938,E2 -27468.938} C_VEL
LIN {X 0,Y 89.841,Z 952.788,A -85,B 0,C 180,E1 -27477.985,E2 -27477.985} C_VEL
LIN {X 0,Y 95.513,Z 949.152,A -85,B 0,C 180,E1 -27486.053,E2 -27486.053} C_VEL
LIN {X 0,Y 100.983,Z 945.32,A -85,B 0,C 180,E1 -27491.38,E2 -27491.38} C_VEL
LIN {X 0,Y 107.318,Z 940.481,A -85,B 0,C 180,E1 -27496.076,E2 -27496.076} C_VEL
LIN {X 0,Y 115.676,Z 933.397,A -85,B 0,C 180,E1 -27500.763,E2 -27500.763} C_VEL
LIN {X 0,Y 123.541,Z 925.85,A -85,B 0,C 180,E1 -27504.151,E2 -27504.151} C_VEL
LIN {X 0,Y 131.892,Z 916.622,A -85,B 0,C 180,E1 -27507.053,E2 -27507.053} C_VEL
LIN {X 0,Y 139.096,Z 907.215,A -85,B 0,C 180,E1 -27509.189,E2 -27509.189} C_VEL
LIN {X 0,Y 139.867,Z 906.109,A -85,B 0,C 180,E1 -27509.382,E2 -27509.382} C_VEL
LIN {X 0,Y 142.69,Z 901.552,A -85,B 0,C 180,E1 -27510.374,E2 -27510.374} C_VEL
LIN {X 0,Y 146.215,Z 893.969,A -85,B 0,C 180,E1 -27512.506,E2 -27512.506} C_VEL
LIN {X 0,Y 149.416,Z 886.047,A -85,B 0,C 180,E1 -27514.457,E2 -27514.457} C_VEL
LIN {X 0,Y 151.627,Z 880.908,A -85,B 0,C 180,E1 -27515.173,E2 -27515.173} C_VEL
LIN {X 0,Y 156.646,Z 868.607,A -85,B 0,C 180,E1 -27516.049,E2 -27516.049} C_VEL
LIN {X 0,Y 160.62,Z 855.349,A -85,B 0,C 180,E1 -27516.75,E2 -27516.75} C_VEL
LIN {X 0,Y 162.664,Z 842.743,A -85,B 0,C 180,E1 -27517.84,E2 -27517.84} C_VEL
LIN {X 0,Y 162.883,Z 840.457,A -85,B 0,C 180,E1 -27518.069,E2 -27518.069} C_VEL
LIN {X 0,Y 162.195,Z 834.623,A -85,B 0,C 180,E1 -27521.037,E2 -27521.037} C_VEL
LIN {X 0,Y 161.663,Z 830.064,A -85,B 0,C 180,E1 -27524.412,E2 -27524.412} C_VEL
LIN {X 0,Y 161.579,Z 827.017,A -85,B 0,C 180,E1 -27528.284,E2 -27528.284} C_VEL
LIN {X 0,Y 161.794,Z 826.944,A -85,B 0,C 180,E1 -27531.256,E2 -27531.256} C_VEL
LIN {X 0,Y 162.283,Z 827.66,A -85,B 0,C 180,E1 -27533.909,E2 -27533.909} C_VEL
LIN {X 0,Y 163.445,Z 831.172,A -85,B 0,C 180,E1 -27537.865,E2 -27537.865} C_VEL
LIN {X 0,Y 164.238,Z 834.283,A -85,B 0,C 180,E1 -27540.099,E2 -27540.099} C_VEL
LIN {X 0,Y 161.656,Z 847.292,A -85,B 0,C 180,E1 -27540.988,E2 -27540.988} C_VEL
LIN {X 0,Y 158.092,Z 859.299,A -85,B 0,C 180,E1 -27542.091,E2 -27542.091} C_VEL
LIN {X 0,Y 153.98,Z 869.657,A -85,B 0,C 180,E1 -27543.291,E2 -27543.291} C_VEL
LIN {X 0,Y 148.149,Z 881.181,A -85,B 0,C 180,E1 -27545.039,E2 -27545.039} C_VEL
LIN {X 0,Y 141.628,Z 891.454,A -85,B 0,C 180,E1 -27547.08,E2 -27547.08} C_VEL
LIN {X 0,Y 135.297,Z 899.787,A -85,B 0,C 180,E1 -27549.294,E2 -27549.294} C_VEL
LIN {X 0,Y 128.166,Z 907.693,A -85,B 0,C 180,E1 -27552.019,E2 -27552.019} C_VEL
LIN {X 0,Y 120.329,Z 915.024,A -85,B 0,C 180,E1 -27555.504,E2 -27555.504} C_VEL
LIN {X 0,Y 112.058,Z 921.414,A -85,B 0,C 180,E1 -27559.836,E2 -27559.836} C_VEL
LIN {X 0,Y 104.374,Z 926.344,A -85,B 0,C 180,E1 -27564.906,E2 -27564.906} C_VEL
LIN {X 0,Y 97.757,Z 929.755,A -85,B 0,C 180,E1 -27570.39,E2 -27570.39} C_VEL
LIN {X 0,Y 93.752,Z 931.37,A -85,B 0,C 180,E1 -27574.464,E2 -27574.464} C_VEL
LIN {X 0,Y 90.241,Z 932.508,A -85,B 0,C 180,E1 -27578.86,E2 -27578.86} C_VEL
LIN {X 0,Y 87.247,Z 933.149,A -85,B 0,C 180,E1 -27583.543,E2 -27583.543} C_VEL
LIN {X 0,Y 84.774,Z 933.307,A -85,B 0,C 180,E1 -27588.464,E2 -27588.464} C_VEL
LIN {X 0,Y 82.937,Z 933.024,A -85,B 0,C 180,E1 -27593.627,E2 -27593.627} C_VEL
LIN {X 0,Y 81.592,Z 932.141,A -85,B 0,C 180,E1 -27599.472,E2 -27599.472} C_VEL
LIN {X 0,Y 81.058,Z 931.022,A -85,B 0,C 180,E1 -27604.318,E2 -27604.318} C_VEL
LIN {X 0,Y 81.302,Z 928.474,A -85,B 0,C 180,E1 -27611.969,E2 -27611.969} C_VEL
LIN {X 0,Y 83.005,Z 924.481,A -85,B 0,C 180,E1 -27620.258,E2 -27620.258} C_VEL
LIN {X 0,Y 85.843,Z 919.489,A -85,B 0,C 180,E1 -27627.661,E2 -27627.661} C_VEL
LIN {X 0,Y 89.757,Z 913.14,A -85,B 0,C 180,E1 -27634.498,E2 -27634.498} C_VEL
LIN {X 0,Y 94.556,Z 905.261,A -85,B 0,C 180,E1 -27640.715,E2 -27640.715} C_VEL
LIN {X 0,Y 99.194,Z 897.237,A -85,B 0,C 180,E1 -27645.414,E2 -27645.414} C_VEL
LIN {X 0,Y 104.234,Z 887.515,A -85,B 0,C 180,E1 -27649.708,E2 -27649.708} C_VEL
LIN {X 0,Y 109.103,Z 876.697,A -85,B 0,C 180,E1 -27653.244,E2 -27653.244} C_VEL
LIN {X 0,Y 113.583,Z 864.75,A -85,B 0,C 180,E1 -27656.165,E2 -27656.165} C_VEL
LIN {X 0,Y 117.308,Z 852.072,A -85,B 0,C 180,E1 -27658.4,E2 -27658.4} C_VEL
LIN {X 0,Y 120.132,Z 838.681,A -85,B 0,C 180,E1 -27660.12,E2 -27660.12} C_VEL
LIN {X 0,Y 121.828,Z 825.143,A -85,B 0,C 180,E1 -27661.284,E2 -27661.284} C_VEL
LIN {X 0,Y 123.136,Z 805.458,A -85,B 0,C 180,E1 -27662.499,E2 -27662.499} C_VEL
LIN {X 0,Y 119.536,Z 797.474,A -85,B 0,C 180,E1 -27665.404,E2 -27665.404} C_VEL
LIN {X 0,Y 119.223,Z 797.564,A -85,B 0,C 180,E1 -27665.591,E2 -27665.591} C_VEL
LIN {X 0,Y 114.622,Z 812.419,A -85,B 0,C 180,E1 -27667.002,E2 -27667.002} C_VEL
LIN {X 0,Y 111.266,Z 821.025,A -85,B 0,C 180,E1 -27668.366,E2 -27668.366} C_VEL
LIN {X 0,Y 108.674,Z 826.069,A -85,B 0,C 180,E1 -27669.683,E2 -27669.683} C_VEL
LIN {X 0,Y 106.471,Z 829.488,A -85,B 0,C 180,E1 -27670.961,E2 -27670.961} C_VEL
LIN {X 0,Y 101.931,Z 840.443,A -85,B 0,C 180,E1 -27672.634,E2 -27672.634} C_VEL
LIN {X 0,Y 97.966,Z 847.541,A -85,B 0,C 180,E1 -27674.355,E2 -27674.355} C_VEL
LIN {X 0,Y 95.437,Z 850.969,A -85,B 0,C 180,E1 -27675.79,E2 -27675.79} C_VEL
LIN {X 0,Y 92.47,Z 853.948,A -85,B 0,C 180,E1 -27678.105,E2 -27678.105} C_VEL
LIN {X 0,Y 90.907,Z 855.37,A -85,B 0,C 180,E1 -27679.543,E2 -27679.543} C_VEL
LIN {X 0,Y 87.634,Z 860.142,A -85,B 0,C 180,E1 -27681.571,E2 -27681.571} C_VEL
LIN {X 0,Y 84.427,Z 863.911,A -85,B 0,C 180,E1 -27684.358,E2 -27684.358} C_VEL
LIN {X 0,Y 82.728,Z 865.39,A -85,B 0,C 180,E1 -27687.282,E2 -27687.282} C_VEL
LIN {X 0,Y 82.267,Z 867.652,A -85,B 0,C 180,E1 -27689.163,E2 -27689.163} C_VEL
LIN {X 0,Y 80.714,Z 881.815,A -85,B 0,C 180,E1 -27696.251,E2 -27696.251} C_VEL
LIN {X 0,Y 80.041,Z 893.249,A -85,B 0,C 180,E1 -27703.418,E2 -27703.418} C_VEL
LIN {X 0,Y 80.486,Z 903.337,A -85,B 0,C 180,E1 -27711.209,E2 -27711.209} C_VEL
LIN {X 0,Y 81.885,Z 910.463,A -85,B 0,C 180,E1 -27717.54,E2 -27717.54} C_VEL
LIN {X 0,Y 84.825,Z 917.693,A -85,B 0,C 180,E1 -27724.752,E2 -27724.752} C_VEL
LIN {X 0,Y 89.015,Z 923.781,A -85,B 0,C 180,E1 -27731.383,E2 -27731.383} C_VEL
LIN {X 0,Y 94.316,Z 928.81,A -85,B 0,C 180,E1 -27737.341,E2 -27737.341} C_VEL
LIN {X 0,Y 100.706,Z 932.956,A -85,B 0,C 180,E1 -27742.571,E2 -27742.571} C_VEL
LIN {X 0,Y 107.936,Z 936.213,A -85,B 0,C 180,E1 -27747.115,E2 -27747.115} C_VEL
LIN {X 0,Y 118.672,Z 939.255,A -85,B 0,C 180,E1 -27752.208,E2 -27752.208} C_VEL
LIN {X 0,Y 119.961,Z 939.519,A -85,B 0,C 180,E1 -27752.71,E2 -27752.71} C_VEL
LIN {X 0,Y 118.709,Z 939.974,A -85,B 0,C 180,E1 -27754.011,E2 -27754.011} C_VEL
LIN {X 0,Y 108.188,Z 940.575,A -85,B 0,C 180,E1 -27758.774,E2 -27758.774} C_VEL
LIN {X 0,Y 103.346,Z 940.652,A -85,B 0,C 180,E1 -27761.57,E2 -27761.57} C_VEL
LIN {X 0,Y 94.903,Z 939.91,A -85,B 0,C 180,E1 -27768.195,E2 -27768.195} C_VEL
LIN {X 0,Y 86.491,Z 937.392,A -85,B 0,C 180,E1 -27779.976,E2 -27779.976} C_VEL
LIN {X 0,Y 81.957,Z 943.444,A -85,B 0,C 180,E1 -27787.294,E2 -27787.294} C_VEL
LIN {X 0,Y 79.744,Z 947.885,A -85,B 0,C 180,E1 -27794.661,E2 -27794.661} C_VEL
LIN {X 0,Y 79.189,Z 950.243,A -85,B 0,C 180,E1 -27799.768,E2 -27799.768} C_VEL
